SPLINE
SPL {X  -148.173, Y  +313.009, Z    +0.000, E1   +35.624, E3 +294907.954}
SPL {X  -159.343, Y  +347.032, Z    +0.000, E1   +21.245, E3 +294911.798}
SPL {X  -161.787, Y  +362.186, Z    +0.000, E1   +13.182, E3 +294912.994}
SPL {X  -162.692, Y  +374.052, Z    +0.000, E1    +6.208, E3 +294912.840}
SPL {X  -162.820, Y  +381.030, Z    +0.000, E1    +1.454, E3 +294913.019}
SPL {X  -162.820, Y  +384.274, Z    +0.000, E1    -1.205, E3 +294912.738}
SPL {X  -162.820, Y  +388.271, Z    +0.000, E1    -5.458, E3 +294912.730}
SPL {X  -162.820, Y  +394.827, Z    +0.000, E1   -13.677, E3 +294912.420}
SPL {X  -162.820, Y  +402.977, Z    +0.000, E1   -24.772, E3 +294912.702}
SPL {X  -162.820, Y  +413.615, Z    +0.000, E1   -37.560, E3 +294912.493}
SPL {X  -162.820, Y  +452.521, Z    +0.000, E1   -56.942, E3 +294926.785}
SPL {X  -162.820, Y  +459.967, Z    +0.000, E1   -57.801, E3 +294932.081}
SPL {X  -162.820, Y  +525.017, Z    +0.000, E1   -58.379, E3 +295000.199}
ENDSPLINE

SPLINE
SPL {X  -162.820, Y  +515.796, Z    +0.000, E1   -54.952, E3 +295009.306}
ENDSPLINE

SPLINE
SPL {X  -162.820, Y  +522.537, Z    +0.000, E1   -55.218, E3 +295017.481}
SPL {X  -162.820, Y  +529.742, Z    +0.000, E1   -55.146, E3 +295028.408}
SPL {X  -162.820, Y  +538.383, Z    +0.000, E1   -55.306, E3 +295039.860}
SPL {X  -162.820, Y  +544.790, Z    +0.000, E1   -55.066, E3 +295050.660}
SPL {X  -162.820, Y  +552.981, Z    +0.000, E1   -55.286, E3 +295061.122}
SPL {X  -162.820, Y  +560.767, Z    +0.000, E1   -55.137, E3 +295073.431}
SPL {X  -162.820, Y  +570.590, Z    +0.000, E1   -55.270, E3 +295086.765}
SPL {X  -162.820, Y  +580.865, Z    +0.000, E1   -55.132, E3 +295102.722}
SPL {X  -162.820, Y  +591.604, Z    +0.000, E1   -55.202, E3 +295117.659}
SPL {X  -162.820, Y  +600.465, Z    +0.000, E1   -55.218, E3 +295130.447}
SPL {X  -162.820, Y  +609.951, Z    +0.000, E1   -55.211, E3 +295144.195}
SPL {X  -162.820, Y  +618.960, Z    +0.000, E1   -55.186, E3 +295157.415}
SPL {X  -162.820, Y  +627.322, Z    +0.000, E1   -55.201, E3 +295169.350}
SPL {X  -162.820, Y  +634.693, Z    +0.000, E1   -55.198, E3 +295180.067}
SPL {X  -162.820, Y  +642.452, Z    +0.000, E1   -55.141, E3 +295191.674}
SPL {X  -162.820, Y  +649.370, Z    +0.000, E1   -55.160, E3 +295201.530}
SPL {X  -162.820, Y  +658.542, Z    +0.000, E1   -55.251, E3 +295214.409}
SPL {X  -162.820, Y  +668.534, Z    +0.000, E1   -55.182, E3 +295229.204}
SPL {X  -162.763, Y  +677.803, Z    +0.000, E1   -55.175, E3 +295242.710}
SPL {X  -162.314, Y  +686.325, Z    +0.000, E1   -55.173, E3 +295254.990}
SPL {X  -161.784, Y  +691.841, Z    +0.000, E1   -55.010, E3 +295263.952}
SPL {X  -161.070, Y  +697.305, Z    +0.000, E1   -54.828, E3 +295273.030}
SPL {X  -159.751, Y  +704.965, Z    +0.000, E1   -54.697, E3 +295285.016}
SPL {X  -158.271, Y  +711.718, Z    +0.000, E1   -54.504, E3 +295295.825}
SPL {X  -157.115, Y  +716.223, Z    +0.000, E1   -54.227, E3 +295304.017}
SPL {X  -155.622, Y  +721.376, Z    +0.000, E1   -53.849, E3 +295313.617}
SPL {X  -153.323, Y  +728.294, Z    +0.000, E1   -53.618, E3 +295325.090}
SPL {X  -150.606, Y  +735.372, Z    +0.000, E1   -53.091, E3 +295338.086}
SPL {X  -148.712, Y  +739.795, Z    +0.000, E1   -52.656, E3 +295346.649}
SPL {X  -146.885, Y  +743.751, Z    +0.000, E1   -52.544, E3 +295352.922}
SPL {X  -144.373, Y  +748.778, Z    +0.000, E1   -52.887, E3 +295358.385}
SPL {X  -137.947, Y  +759.993, Z    +0.000, E1   -55.381, E3 +295361.495}
SPL {X  -123.111, Y  +780.056, Z    +0.000, E1   -48.144, E3 +295460.630}
ENDSPLINE

SPLINE
SPL {X  -146.599, Y  +744.345, Z    +0.000, E1   -36.661, E3 +295545.633}
SPL {X  -158.886, Y  +709.076, Z    +0.000, E1   -22.176, E3 +295549.505}
SPL {X  -161.886, Y  +690.913, Z    +0.000, E1   -12.672, E3 +295554.140}
SPL {X  -162.573, Y  +682.458, Z    +0.000, E1    -7.683, E3 +295553.641}
SPL {X  -162.817, Y  +674.426, Z    +0.000, E1    -2.573, E3 +295553.359}
SPL {X  -162.820, Y  +670.554, Z    +0.000, E1    +0.472, E3 +295552.983}
SPL {X  -162.820, Y  +667.789, Z    +0.000, E1    +3.144, E3 +295553.005}
SPL {X  -162.820, Y  +664.083, Z    +0.000, E1    +7.387, E3 +295552.897}
SPL {X  -162.820, Y  +659.344, Z    +0.000, E1   +13.535, E3 +295552.460}
SPL {X  -162.820, Y  +653.403, Z    +0.000, E1   +21.415, E3 +295552.875}
SPL {X  -162.820, Y  +642.162, Z    +0.000, E1   +35.510, E3 +295552.187}
SPL {X  -162.820, Y  +598.675, Z    +0.000, E1   +56.845, E3 +295569.500}
SPL {X  -162.820, Y  +543.175, Z    +0.000, E1   +54.504, E3 +295645.354}
SPL {X  -162.820, Y  +538.115, Z    +0.000, E1   +53.658, E3 +295658.406}
SPL {X  -162.820, Y  +527.429, Z    +0.000, E1   +53.760, E3 +295674.135}
SPL {X  -162.820, Y  +518.365, Z    +0.000, E1   +53.683, E3 +295688.393}
SPL {X  -162.820, Y  +510.654, Z    +0.000, E1   +53.658, E3 +295700.392}
SPL {X  -162.820, Y  +501.304, Z    +0.000, E1   +53.758, E3 +295714.081}
SPL {X  -162.820, Y  +493.008, Z    +0.000, E1   +53.586, E3 +295727.856}
SPL {X  -162.820, Y  +484.615, Z    +0.000, E1   +53.726, E3 +295739.787}
ENDSPLINE

SPLINE
SPL {X  -162.820, Y  +492.996, Z    +0.000, E1   +49.430, E3 +295752.333}
ENDSPLINE

SPLINE
SPL {X  -162.820, Y  +486.578, Z    +0.000, E1   +49.194, E3 +295765.136}
SPL {X  -162.820, Y  +476.731, Z    +0.000, E1   +50.039, E3 +295777.558}
SPL {X  -162.820, Y  +466.442, Z    +0.000, E1   +50.873, E3 +295790.227}
SPL {X  -162.820, Y  +458.457, Z    +0.000, E1   +51.401, E3 +295800.366}
SPL {X  -162.820, Y  +452.070, Z    +0.000, E1   +52.035, E3 +295807.002}
SPL {X  -162.820, Y  +442.466, Z    +0.000, E1   +52.743, E3 +295818.214}
SPL {X  -162.820, Y  +429.602, Z    +0.000, E1   +53.907, E3 +295830.916}
SPL {X  -162.820, Y  +419.900, Z    +0.000, E1   +54.598, E3 +295841.168}
SPL {X  -162.820, Y  +411.092, Z    +0.000, E1   +54.552, E3 +295854.688}
SPL {X  -162.820, Y  +400.244, Z    +0.000, E1   +54.630, E3 +295870.155}
SPL {X  -162.820, Y  +392.496, Z    +0.000, E1   +54.734, E3 +295880.856}
SPL {X  -162.820, Y  +387.085, Z    +0.000, E1   +54.699, E3 +295889.083}
SPL {X  -162.820, Y  +380.650, Z    +0.000, E1   +54.601, E3 +295899.179}
SPL {X  -162.727, Y  +374.992, Z    +0.000, E1   +54.549, E3 +295907.861}
SPL {X  -162.373, Y  +368.447, Z    +0.000, E1   +54.597, E3 +295917.293}
SPL {X  -161.939, Y  +363.587, Z    +0.000, E1   +54.355, E3 +295925.905}
SPL {X  -161.062, Y  +356.641, Z    +0.000, E1   +54.440, E3 +295935.778}
SPL {X  -159.761, Y  +349.086, Z    +0.000, E1   +54.132, E3 +295948.799}
SPL {X  -158.033, Y  +341.310, Z    +0.000, E1   +53.819, E3 +295962.189}
SPL {X  -156.195, Y  +334.528, Z    +0.000, E1   +53.534, E3 +295973.755}
SPL {X  -154.120, Y  +327.988, Z    +0.000, E1   +53.171, E3 +295985.612}
SPL {X  -151.310, Y  +320.369, Z    +0.000, E1   +52.706, E3 +295999.327}
SPL {X  -148.923, Y  +314.679, Z    +0.000, E1   +52.172, E3 +296010.411}
SPL {X  -146.846, Y  +310.168, Z    +0.000, E1   +51.697, E3 +296019.473}
SPL {X  -140.627, Y  +298.437, Z    +0.000, E1   +54.251, E3 +296023.731}
SPL {X  -122.064, Y  +272.747, Z    +0.000, E1   +48.156, E3 +296129.257}
ENDSPLINE

SPLINE
SPL {X  -148.173, Y  +313.009, Z    +0.000, E1   +35.624, E3 +296212.302}
SPL {X  -158.289, Y  +342.356, Z    +0.000, E1   +23.452, E3 +296215.292}
SPL {X  -161.301, Y  +358.312, Z    +0.000, E1   +15.384, E3 +296217.249}
SPL {X  -162.692, Y  +374.052, Z    +0.000, E1    +6.208, E3 +296217.188}
SPL {X  -162.820, Y  +381.030, Z    +0.000, E1    +1.454, E3 +296217.366}
SPL {X  -162.820, Y  +384.274, Z    +0.000, E1    -1.205, E3 +296217.086}
SPL {X  -162.820, Y  +388.271, Z    +0.000, E1    -5.458, E3 +296217.078}
SPL {X  -162.820, Y  +394.827, Z    +0.000, E1   -13.677, E3 +296216.768}
SPL {X  -162.820, Y  +402.977, Z    +0.000, E1   -24.772, E3 +296217.050}
SPL {X  -162.820, Y  +413.615, Z    +0.000, E1   -37.560, E3 +296216.841}
SPL {X  -162.820, Y  +456.390, Z    +0.000, E1   -57.415, E3 +296233.882}
SPL {X  -162.820, Y  +525.017, Z    +0.000, E1   -58.379, E3 +296304.547}
ENDSPLINE

SPLINE
SPL {X  -162.820, Y  +520.266, Z    +0.000, E1   -55.155, E3 +296319.039}
ENDSPLINE

SPLINE
SPL {X  -162.820, Y  +529.742, Z    +0.000, E1   -55.146, E3 +296332.755}
SPL {X  -162.820, Y  +538.383, Z    +0.000, E1   -55.306, E3 +296344.208}
SPL {X  -162.820, Y  +544.790, Z    +0.000, E1   -55.066, E3 +296355.008}
SPL {X  -162.820, Y  +555.105, Z    +0.000, E1   -55.222, E3 +296369.128}
SPL {X  -162.820, Y  +563.355, Z    +0.000, E1   -55.172, E3 +296381.195}
SPL {X  -162.820, Y  +570.590, Z    +0.000, E1   -55.270, E3 +296391.113}
SPL {X  -162.820, Y  +580.865, Z    +0.000, E1   -55.132, E3 +296407.070}
SPL {X  -162.820, Y  +591.604, Z    +0.000, E1   -55.202, E3 +296422.007}
SPL {X  -162.820, Y  +600.465, Z    +0.000, E1   -55.218, E3 +296434.795}
SPL {X  -162.820, Y  +609.951, Z    +0.000, E1   -55.211, E3 +296448.543}
SPL {X  -162.820, Y  +618.960, Z    +0.000, E1   -55.186, E3 +296461.763}
SPL {X  -162.820, Y  +627.322, Z    +0.000, E1   -55.201, E3 +296473.698}
SPL {X  -162.820, Y  +634.693, Z    +0.000, E1   -55.198, E3 +296484.415}
SPL {X  -162.820, Y  +642.452, Z    +0.000, E1   -55.141, E3 +296496.021}
SPL {X  -162.820, Y  +649.370, Z    +0.000, E1   -55.160, E3 +296505.878}
SPL {X  -162.820, Y  +658.542, Z    +0.000, E1   -55.251, E3 +296518.757}
SPL {X  -162.820, Y  +668.534, Z    +0.000, E1   -55.182, E3 +296533.552}
SPL {X  -162.763, Y  +677.803, Z    +0.000, E1   -55.175, E3 +296547.058}
SPL {X  -162.084, Y  +688.960, Z    +0.000, E1   -55.150, E3 +296563.513}
SPL {X  -161.070, Y  +697.305, Z    +0.000, E1   -54.828, E3 +296577.378}
SPL {X  -159.751, Y  +704.965, Z    +0.000, E1   -54.697, E3 +296589.364}
SPL {X  -158.271, Y  +711.718, Z    +0.000, E1   -54.504, E3 +296600.173}
SPL {X  -157.115, Y  +716.223, Z    +0.000, E1   -54.227, E3 +296608.364}
SPL {X  -155.622, Y  +721.376, Z    +0.000, E1   -53.849, E3 +296617.964}
SPL {X  -153.323, Y  +728.294, Z    +0.000, E1   -53.618, E3 +296629.437}
SPL {X  -150.606, Y  +735.372, Z    +0.000, E1   -53.091, E3 +296642.434}
SPL {X  -148.712, Y  +739.795, Z    +0.000, E1   -52.656, E3 +296650.997}
SPL {X  -146.885, Y  +743.751, Z    +0.000, E1   -52.544, E3 +296657.270}
SPL {X  -144.373, Y  +748.778, Z    +0.000, E1   -52.887, E3 +296662.733}
SPL {X  -137.947, Y  +759.993, Z    +0.000, E1   -55.381, E3 +296665.842}
SPL {X  -123.111, Y  +780.056, Z    +0.000, E1   -48.144, E3 +296764.978}
ENDSPLINE

SPLINE
SPL {X  -146.599, Y  +744.345, Z    +0.000, E1   -36.661, E3 +296849.981}
SPL {X  -158.886, Y  +709.076, Z    +0.000, E1   -22.176, E3 +296853.853}
SPL {X  -161.886, Y  +690.913, Z    +0.000, E1   -12.672, E3 +296858.488}
SPL {X  -162.700, Y  +679.756, Z    +0.000, E1    -6.060, E3 +296857.697}
SPL {X  -162.820, Y  +673.439, Z    +0.000, E1    -1.797, E3 +296857.799}
SPL {X  -162.820, Y  +670.554, Z    +0.000, E1    +0.472, E3 +296857.331}
SPL {X  -162.820, Y  +667.789, Z    +0.000, E1    +3.144, E3 +296857.353}
SPL {X  -162.820, Y  +664.083, Z    +0.000, E1    +7.387, E3 +296857.244}
SPL {X  -162.820, Y  +659.344, Z    +0.000, E1   +13.535, E3 +296856.808}
SPL {X  -162.820, Y  +653.403, Z    +0.000, E1   +21.415, E3 +296857.223}
SPL {X  -162.820, Y  +642.162, Z    +0.000, E1   +35.510, E3 +296856.535}
SPL {X  -162.820, Y  +598.675, Z    +0.000, E1   +56.845, E3 +296873.848}
SPL {X  -162.820, Y  +542.287, Z    +0.000, E1   +54.257, E3 +296952.751}
SPL {X  -162.820, Y  +533.839, Z    +0.000, E1   +53.682, E3 +296969.172}
SPL {X  -162.820, Y  +525.300, Z    +0.000, E1   +53.701, E3 +296981.947}
SPL {X  -162.820, Y  +518.365, Z    +0.000, E1   +53.683, E3 +296992.741}
SPL {X  -162.820, Y  +508.465, Z    +0.000, E1   +53.706, E3 +297007.956}
SPL {X  -162.820, Y  +499.206, Z    +0.000, E1   +53.779, E3 +297021.395}
SPL {X  -162.820, Y  +493.008, Z    +0.000, E1   +53.586, E3 +297032.204}
SPL {X  -162.820, Y  +485.759, Z    +0.000, E1   +53.138, E3 +297046.211}
ENDSPLINE

SPLINE
SPL {X  -162.820, Y  +494.645, Z    +0.000, E1   +48.544, E3 +297058.687}
ENDSPLINE

SPLINE
SPL {X  -162.820, Y  +486.578, Z    +0.000, E1   +49.194, E3 +297069.483}
SPL {X  -162.820, Y  +476.731, Z    +0.000, E1   +50.039, E3 +297081.906}
SPL {X  -162.820, Y  +466.442, Z    +0.000, E1   +50.873, E3 +297094.575}
SPL {X  -162.820, Y  +458.457, Z    +0.000, E1   +51.401, E3 +297104.714}
SPL {X  -162.820, Y  +452.070, Z    +0.000, E1   +52.035, E3 +297111.349}
SPL {X  -162.820, Y  +442.466, Z    +0.000, E1   +52.743, E3 +297122.562}
SPL {X  -162.820, Y  +429.602, Z    +0.000, E1   +53.907, E3 +297135.264}
SPL {X  -162.820, Y  +419.900, Z    +0.000, E1   +54.598, E3 +297145.516}
SPL {X  -162.820, Y  +411.092, Z    +0.000, E1   +54.552, E3 +297159.036}
SPL {X  -162.820, Y  +400.244, Z    +0.000, E1   +54.630, E3 +297174.503}
SPL {X  -162.820, Y  +389.249, Z    +0.000, E1   +54.752, E3 +297190.082}
SPL {X  -162.799, Y  +377.862, Z    +0.000, E1   +54.622, E3 +297207.712}
SPL {X  -162.373, Y  +368.447, Z    +0.000, E1   +54.597, E3 +297221.641}
SPL {X  -161.939, Y  +363.587, Z    +0.000, E1   +54.355, E3 +297230.253}
SPL {X  -161.062, Y  +356.641, Z    +0.000, E1   +54.440, E3 +297240.126}
SPL {X  -159.761, Y  +349.086, Z    +0.000, E1   +54.132, E3 +297253.147}
SPL {X  -158.451, Y  +343.033, Z    +0.000, E1   +53.828, E3 +297263.824}
SPL {X  -156.619, Y  +335.993, Z    +0.000, E1   +53.639, E3 +297275.470}
SPL {X  -154.959, Y  +330.520, Z    +0.000, E1   +53.198, E3 +297285.895}
SPL {X  -152.785, Y  +324.223, Z    +0.000, E1   +52.975, E3 +297296.568}
SPL {X  -150.663, Y  +318.766, Z    +0.000, E1   +52.574, E3 +297306.601}
SPL {X  -148.923, Y  +314.679, Z    +0.000, E1   +52.172, E3 +297314.759}
SPL {X  -146.846, Y  +310.168, Z    +0.000, E1   +51.697, E3 +297323.820}
SPL {X  -140.627, Y  +298.437, Z    +0.000, E1   +54.251, E3 +297328.079}
SPL {X  -121.787, Y  +272.434, Z    +0.000, E1   +49.053, E3 +297418.440}
ENDSPLINE

SPLINE
SPL {X  -122.346, Y  +273.067, Z    +0.000, E1   +47.776, E3 +297439.631}
SPL {X  -148.173, Y  +313.009, Z    +0.000, E1   +35.624, E3 +297516.650}
SPL {X  -159.343, Y  +347.032, Z    +0.000, E1   +21.245, E3 +297520.494}
SPL {X  -161.787, Y  +362.186, Z    +0.000, E1   +13.182, E3 +297521.689}
SPL {X  -162.692, Y  +374.052, Z    +0.000, E1    +6.208, E3 +297521.535}
SPL {X  -162.820, Y  +382.143, Z    +0.000, E1    +0.693, E3 +297521.670}
SPL {X  -162.820, Y  +385.887, Z    +0.000, E1    -2.819, E3 +297521.342}
SPL {X  -162.820, Y  +389.383, Z    +0.000, E1    -6.871, E3 +297521.409}
SPL {X  -162.820, Y  +393.153, Z    +0.000, E1   -11.600, E3 +297521.303}
SPL {X  -162.820, Y  +400.748, Z    +0.000, E1   -21.791, E3 +297521.094}
SPL {X  -162.820, Y  +413.615, Z    +0.000, E1   -37.560, E3 +297521.189}
SPL {X  -162.820, Y  +456.390, Z    +0.000, E1   -57.415, E3 +297538.230}
SPL {X  -162.820, Y  +525.017, Z    +0.000, E1   -58.379, E3 +297608.895}
ENDSPLINE

SPLINE
SPL {X  -162.820, Y  +520.266, Z    +0.000, E1   -55.155, E3 +297623.387}
ENDSPLINE

SPLINE
SPL {X  -162.820, Y  +529.742, Z    +0.000, E1   -55.146, E3 +297637.103}
SPL {X  -162.820, Y  +538.383, Z    +0.000, E1   -55.306, E3 +297648.555}
SPL {X  -162.820, Y  +544.790, Z    +0.000, E1   -55.066, E3 +297659.356}
SPL {X  -162.820, Y  +552.981, Z    +0.000, E1   -55.286, E3 +297669.818}
SPL {X  -162.820, Y  +560.767, Z    +0.000, E1   -55.137, E3 +297682.126}
SPL {X  -162.820, Y  +570.590, Z    +0.000, E1   -55.270, E3 +297695.461}
SPL {X  -162.820, Y  +577.946, Z    +0.000, E1   -55.110, E3 +297707.098}
SPL {X  -162.820, Y  +583.981, Z    +0.000, E1   -55.057, E3 +297716.181}
SPL {X  -162.820, Y  +591.604, Z    +0.000, E1   -55.202, E3 +297726.355}
SPL {X  -162.820, Y  +600.465, Z    +0.000, E1   -55.218, E3 +297739.143}
SPL {X  -162.820, Y  +609.951, Z    +0.000, E1   -55.211, E3 +297752.891}
SPL {X  -162.820, Y  +618.960, Z    +0.000, E1   -55.186, E3 +297766.111}
SPL {X  -162.820, Y  +627.322, Z    +0.000, E1   -55.201, E3 +297778.046}
SPL {X  -162.820, Y  +634.693, Z    +0.000, E1   -55.198, E3 +297788.763}
SPL {X  -162.820, Y  +642.452, Z    +0.000, E1   -55.141, E3 +297800.369}
SPL {X  -162.820, Y  +652.837, Z    +0.000, E1   -55.281, E3 +297814.637}
SPL {X  -162.820, Y  +660.849, Z    +0.000, E1   -55.101, E3 +297827.186}
SPL {X  -162.820, Y  +668.534, Z    +0.000, E1   -55.182, E3 +297837.900}
SPL {X  -162.763, Y  +677.803, Z    +0.000, E1   -55.175, E3 +297851.406}
SPL {X  -162.084, Y  +688.960, Z    +0.000, E1   -55.150, E3 +297867.861}
SPL {X  -161.070, Y  +697.305, Z    +0.000, E1   -54.828, E3 +297881.726}
SPL {X  -159.751, Y  +704.965, Z    +0.000, E1   -54.697, E3 +297893.712}
SPL {X  -158.271, Y  +711.718, Z    +0.000, E1   -54.504, E3 +297904.521}
SPL {X  -157.115, Y  +716.223, Z    +0.000, E1   -54.227, E3 +297912.712}
SPL {X  -154.825, Y  +723.894, Z    +0.000, E1   -53.830, E3 +297926.252}
SPL {X  -152.160, Y  +731.445, Z    +0.000, E1   -53.336, E3 +297939.795}
SPL {X  -150.059, Y  +736.687, Z    +0.000, E1   -53.023, E3 +297948.961}
SPL {X  -147.746, Y  +741.922, Z    +0.000, E1   -52.631, E3 +297958.668}
SPL {X  -144.373, Y  +748.778, Z    +0.000, E1   -52.887, E3 +297967.081}
SPL {X  -137.947, Y  +759.993, Z    +0.000, E1   -55.381, E3 +297970.190}
SPL {X  -123.111, Y  +780.056, Z    +0.000, E1   -48.144, E3 +298069.326}
ENDSPLINE

SPLINE
SPL {X  -146.599, Y  +744.345, Z    +0.000, E1   -36.661, E3 +298154.329}
SPL {X  -158.886, Y  +709.076, Z    +0.000, E1   -22.176, E3 +298158.201}
SPL {X  -161.886, Y  +690.913, Z    +0.000, E1   -12.672, E3 +298162.835}
SPL {X  -162.700, Y  +679.756, Z    +0.000, E1    -6.060, E3 +298162.045}
SPL {X  -162.820, Y  +673.439, Z    +0.000, E1    -1.797, E3 +298162.146}
SPL {X  -162.820, Y  +670.554, Z    +0.000, E1    +0.472, E3 +298161.679}
SPL {X  -162.820, Y  +667.789, Z    +0.000, E1    +3.144, E3 +298161.701}
SPL {X  -162.820, Y  +664.083, Z    +0.000, E1    +7.387, E3 +298161.592}
SPL {X  -162.820, Y  +659.344, Z    +0.000, E1   +13.535, E3 +298161.156}
SPL {X  -162.820, Y  +653.403, Z    +0.000, E1   +21.415, E3 +298161.571}
SPL {X  -162.820, Y  +642.162, Z    +0.000, E1   +35.510, E3 +298160.883}
SPL {X  -162.820, Y  +598.675, Z    +0.000, E1   +56.845, E3 +298178.195}
SPL {X  -162.820, Y  +543.175, Z    +0.000, E1   +54.504, E3 +298254.050}
SPL {X  -162.820, Y  +538.115, Z    +0.000, E1   +53.658, E3 +298267.101}
SPL {X  -162.820, Y  +527.429, Z    +0.000, E1   +53.760, E3 +298282.831}
SPL {X  -162.820, Y  +518.365, Z    +0.000, E1   +53.683, E3 +298297.089}
SPL {X  -162.820, Y  +510.654, Z    +0.000, E1   +53.658, E3 +298309.088}
SPL {X  -162.820, Y  +501.304, Z    +0.000, E1   +53.758, E3 +298322.776}
SPL {X  -162.820, Y  +493.008, Z    +0.000, E1   +53.586, E3 +298336.552}
SPL {X  -162.820, Y  +484.615, Z    +0.000, E1   +53.726, E3 +298348.482}
ENDSPLINE

SPLINE
SPL {X  -162.820, Y  +492.996, Z    +0.000, E1   +49.430, E3 +298361.028}
ENDSPLINE

SPLINE
SPL {X  -162.820, Y  +486.578, Z    +0.000, E1   +49.194, E3 +298373.831}
SPL {X  -162.820, Y  +476.731, Z    +0.000, E1   +50.039, E3 +298386.254}
SPL {X  -162.820, Y  +466.442, Z    +0.000, E1   +50.873, E3 +298398.922}
SPL {X  -162.820, Y  +455.624, Z    +0.000, E1   +51.698, E3 +298411.994}
SPL {X  -162.820, Y  +444.568, Z    +0.000, E1   +52.608, E3 +298424.306}
SPL {X  -162.820, Y  +432.435, Z    +0.000, E1   +53.605, E3 +298437.189}
SPL {X  -162.820, Y  +419.875, Z    +0.000, E1   +54.604, E3 +298449.864}
SPL {X  -162.820, Y  +414.181, Z    +0.000, E1   +54.446, E3 +298459.298}
SPL {X  -162.820, Y  +407.616, Z    +0.000, E1   +54.585, E3 +298468.132}
SPL {X  -162.820, Y  +400.244, Z    +0.000, E1   +54.630, E3 +298478.851}
SPL {X  -162.820, Y  +389.249, Z    +0.000, E1   +54.752, E3 +298494.430}
SPL {X  -162.820, Y  +380.650, Z    +0.000, E1   +54.601, E3 +298507.875}
SPL {X  -162.727, Y  +374.992, Z    +0.000, E1   +54.549, E3 +298516.557}
SPL {X  -162.373, Y  +368.447, Z    +0.000, E1   +54.597, E3 +298525.989}
SPL {X  -161.939, Y  +363.587, Z    +0.000, E1   +54.355, E3 +298534.601}
SPL {X  -161.062, Y  +356.641, Z    +0.000, E1   +54.440, E3 +298544.474}
SPL {X  -159.761, Y  +349.086, Z    +0.000, E1   +54.132, E3 +298557.495}
SPL {X  -158.033, Y  +341.310, Z    +0.000, E1   +53.819, E3 +298570.885}
SPL {X  -155.608, Y  +332.578, Z    +0.000, E1   +53.425, E3 +298586.156}
SPL {X  -152.785, Y  +324.223, Z    +0.000, E1   +52.975, E3 +298600.916}
SPL {X  -150.663, Y  +318.766, Z    +0.000, E1   +52.574, E3 +298610.949}
SPL {X  -148.923, Y  +314.679, Z    +0.000, E1   +52.172, E3 +298619.107}
SPL {X  -146.846, Y  +310.168, Z    +0.000, E1   +51.697, E3 +298628.168}
SPL {X  -140.627, Y  +298.437, Z    +0.000, E1   +54.251, E3 +298632.427}
SPL {X  -122.064, Y  +272.747, Z    +0.000, E1   +48.156, E3 +298737.952}
ENDSPLINE

SPLINE
SPL {X  -148.173, Y  +313.009, Z    +0.000, E1   +35.624, E3 +298820.998}
SPL {X  -159.343, Y  +347.032, Z    +0.000, E1   +21.245, E3 +298824.842}
SPL {X  -162.355, Y  +368.197, Z    +0.000, E1    +9.799, E3 +298826.010}
SPL {X  -162.819, Y  +380.071, Z    +0.000, E1    +2.240, E3 +298826.005}
SPL {X  -162.820, Y  +384.274, Z    +0.000, E1    -1.205, E3 +298825.781}
SPL {X  -162.820, Y  +388.271, Z    +0.000, E1    -5.458, E3 +298825.774}
SPL {X  -162.820, Y  +394.827, Z    +0.000, E1   -13.677, E3 +298825.464}
SPL {X  -162.820, Y  +402.977, Z    +0.000, E1   -24.772, E3 +298825.746}
SPL {X  -162.820, Y  +413.615, Z    +0.000, E1   -37.560, E3 +298825.536}
SPL {X  -162.820, Y  +456.390, Z    +0.000, E1   -57.415, E3 +298842.578}
SPL {X  -162.820, Y  +525.017, Z    +0.000, E1   -58.379, E3 +298913.242}
ENDSPLINE

SPLINE
SPL {X  -162.820, Y  +515.796, Z    +0.000, E1   -54.952, E3 +298922.349}
ENDSPLINE

SPLINE
SPL {X  -162.820, Y  +522.537, Z    +0.000, E1   -55.218, E3 +298930.524}
SPL {X  -162.820, Y  +529.742, Z    +0.000, E1   -55.146, E3 +298941.451}
SPL {X  -162.820, Y  +538.383, Z    +0.000, E1   -55.306, E3 +298952.903}
SPL {X  -162.820, Y  +544.790, Z    +0.000, E1   -55.066, E3 +298963.703}
SPL {X  -162.820, Y  +555.105, Z    +0.000, E1   -55.222, E3 +298977.824}
SPL {X  -162.820, Y  +563.355, Z    +0.000, E1   -55.172, E3 +298989.891}
SPL {X  -162.820, Y  +570.590, Z    +0.000, E1   -55.270, E3 +298999.808}
SPL {X  -162.820, Y  +580.865, Z    +0.000, E1   -55.132, E3 +299015.765}
SPL {X  -162.820, Y  +594.246, Z    +0.000, E1   -55.310, E3 +299033.964}
SPL {X  -162.820, Y  +601.811, Z    +0.000, E1   -55.027, E3 +299046.492}
SPL {X  -162.820, Y  +609.951, Z    +0.000, E1   -55.211, E3 +299057.238}
SPL {X  -162.820, Y  +618.960, Z    +0.000, E1   -55.186, E3 +299070.459}
SPL {X  -162.820, Y  +627.322, Z    +0.000, E1   -55.201, E3 +299082.394}
SPL {X  -162.820, Y  +634.693, Z    +0.000, E1   -55.198, E3 +299093.110}
SPL {X  -162.820, Y  +642.452, Z    +0.000, E1   -55.141, E3 +299104.717}
SPL {X  -162.820, Y  +649.370, Z    +0.000, E1   -55.160, E3 +299114.574}
SPL {X  -162.820, Y  +658.542, Z    +0.000, E1   -55.251, E3 +299127.452}
SPL {X  -162.820, Y  +671.259, Z    +0.000, E1   -55.266, E3 +299145.830}
SPL {X  -162.498, Y  +683.731, Z    +0.000, E1   -55.157, E3 +299164.539}
SPL {X  -161.784, Y  +691.841, Z    +0.000, E1   -55.010, E3 +299176.996}
SPL {X  -161.070, Y  +697.305, Z    +0.000, E1   -54.828, E3 +299186.074}
SPL {X  -159.751, Y  +704.965, Z    +0.000, E1   -54.697, E3 +299198.060}
SPL {X  -158.271, Y  +711.718, Z    +0.000, E1   -54.504, E3 +299208.868}
SPL {X  -157.115, Y  +716.223, Z    +0.000, E1   -54.227, E3 +299217.060}
SPL {X  -154.825, Y  +723.894, Z    +0.000, E1   -53.830, E3 +299230.600}
SPL {X  -152.160, Y  +731.445, Z    +0.000, E1   -53.336, E3 +299244.142}
SPL {X  -150.059, Y  +736.687, Z    +0.000, E1   -53.023, E3 +299253.308}
SPL {X  -147.746, Y  +741.922, Z    +0.000, E1   -52.631, E3 +299263.016}
SPL {X  -144.373, Y  +748.778, Z    +0.000, E1   -52.887, E3 +299271.428}
SPL {X  -137.947, Y  +759.993, Z    +0.000, E1   -55.381, E3 +299274.538}
SPL {X  -123.111, Y  +780.056, Z    +0.000, E1   -48.144, E3 +299373.674}
ENDSPLINE

SPLINE
SPL {X  -146.599, Y  +744.345, Z    +0.000, E1   -36.661, E3 +299458.677}
SPL {X  -157.185, Y  +715.965, Z    +0.000, E1   -25.340, E3 +299461.727}
SPL {X  -159.997, Y  +703.690, Z    +0.000, E1   -19.457, E3 +299463.055}
SPL {X  -161.886, Y  +690.913, Z    +0.000, E1   -12.672, E3 +299467.183}
SPL {X  -162.700, Y  +679.756, Z    +0.000, E1    -6.060, E3 +299466.392}
SPL {X  -162.820, Y  +673.439, Z    +0.000, E1    -1.797, E3 +299466.494}
SPL {X  -162.820, Y  +670.554, Z    +0.000, E1    +0.472, E3 +299466.027}
SPL {X  -162.820, Y  +667.789, Z    +0.000, E1    +3.144, E3 +299466.048}
SPL {X  -162.820, Y  +664.083, Z    +0.000, E1    +7.387, E3 +299465.940}
SPL {X  -162.820, Y  +659.344, Z    +0.000, E1   +13.535, E3 +299465.504}
SPL {X  -162.820, Y  +653.403, Z    +0.000, E1   +21.415, E3 +299465.918}
SPL {X  -162.820, Y  +642.162, Z    +0.000, E1   +35.510, E3 +299465.231}
SPL {X  -162.820, Y  +598.675, Z    +0.000, E1   +56.845, E3 +299482.543}
SPL {X  -162.820, Y  +543.175, Z    +0.000, E1   +54.504, E3 +299558.398}
SPL {X  -162.820, Y  +538.115, Z    +0.000, E1   +53.658, E3 +299571.449}
SPL {X  -162.820, Y  +527.429, Z    +0.000, E1   +53.760, E3 +299587.179}
SPL {X  -162.820, Y  +518.365, Z    +0.000, E1   +53.683, E3 +299601.437}
SPL {X  -162.820, Y  +510.654, Z    +0.000, E1   +53.658, E3 +299613.436}
SPL {X  -162.820, Y  +501.304, Z    +0.000, E1   +53.758, E3 +299627.124}
SPL {X  -162.820, Y  +493.008, Z    +0.000, E1   +53.586, E3 +299640.899}
SPL {X  -162.820, Y  +484.615, Z    +0.000, E1   +53.726, E3 +299652.830}
ENDSPLINE

SPLINE
SPL {X  -162.820, Y  +492.996, Z    +0.000, E1   +49.430, E3 +299665.376}
ENDSPLINE

SPLINE
SPL {X  -162.820, Y  +486.578, Z    +0.000, E1   +49.194, E3 +299678.179}
SPL {X  -162.820, Y  +476.731, Z    +0.000, E1   +50.039, E3 +299690.602}
SPL {X  -162.820, Y  +466.442, Z    +0.000, E1   +50.873, E3 +299703.270}
SPL {X  -162.820, Y  +455.624, Z    +0.000, E1   +51.698, E3 +299716.341}
SPL {X  -162.820, Y  +444.568, Z    +0.000, E1   +52.608, E3 +299728.654}
SPL {X  -162.820, Y  +432.435, Z    +0.000, E1   +53.605, E3 +299741.537}
SPL {X  -162.820, Y  +419.875, Z    +0.000, E1   +54.604, E3 +299754.211}
SPL {X  -162.820, Y  +414.181, Z    +0.000, E1   +54.446, E3 +299763.646}
SPL {X  -162.820, Y  +407.616, Z    +0.000, E1   +54.585, E3 +299772.480}
SPL {X  -162.820, Y  +400.244, Z    +0.000, E1   +54.630, E3 +299783.198}
SPL {X  -162.820, Y  +389.249, Z    +0.000, E1   +54.752, E3 +299798.777}
SPL {X  -162.799, Y  +377.862, Z    +0.000, E1   +54.622, E3 +299816.408}
SPL {X  -162.373, Y  +368.447, Z    +0.000, E1   +54.597, E3 +299830.337}
SPL {X  -161.939, Y  +363.587, Z    +0.000, E1   +54.355, E3 +299838.949}
SPL {X  -161.062, Y  +356.641, Z    +0.000, E1   +54.440, E3 +299848.822}
SPL {X  -159.761, Y  +349.086, Z    +0.000, E1   +54.132, E3 +299861.843}
SPL {X  -158.451, Y  +343.033, Z    +0.000, E1   +53.828, E3 +299872.520}
SPL {X  -156.619, Y  +335.993, Z    +0.000, E1   +53.639, E3 +299884.166}
SPL {X  -154.120, Y  +327.988, Z    +0.000, E1   +53.171, E3 +299898.656}
SPL {X  -151.310, Y  +320.369, Z    +0.000, E1   +52.706, E3 +299912.370}
SPL {X  -148.923, Y  +314.679, Z    +0.000, E1   +52.172, E3 +299923.455}
SPL {X  -146.846, Y  +310.168, Z    +0.000, E1   +51.697, E3 +299932.516}
SPL {X  -140.627, Y  +298.437, Z    +0.000, E1   +54.251, E3 +299936.775}
SPL {X  -122.064, Y  +272.747, Z    +0.000, E1   +48.156, E3 +300042.300}
ENDSPLINE

SPLINE
SPL {X  -148.173, Y  +313.009, Z    +0.000, E1   +35.624, E3 +300125.346}
SPL {X  -159.343, Y  +347.032, Z    +0.000, E1   +21.245, E3 +300129.189}
SPL {X  -162.355, Y  +368.197, Z    +0.000, E1    +9.799, E3 +300130.358}
SPL {X  -162.819, Y  +380.071, Z    +0.000, E1    +2.240, E3 +300130.353}
SPL {X  -162.820, Y  +383.414, Z    +0.000, E1    -0.499, E3 +300130.316}
SPL {X  -162.820, Y  +385.887, Z    +0.000, E1    -2.819, E3 +300130.038}
SPL {X  -162.820, Y  +389.383, Z    +0.000, E1    -6.871, E3 +300130.105}
SPL {X  -162.820, Y  +393.153, Z    +0.000, E1   -11.600, E3 +300129.999}
SPL {X  -162.820, Y  +400.748, Z    +0.000, E1   -21.791, E3 +300129.790}
SPL {X  -162.820, Y  +413.615, Z    +0.000, E1   -37.560, E3 +300129.884}
SPL {X  -162.820, Y  +456.390, Z    +0.000, E1   -57.415, E3 +300146.926}
SPL {X  -162.820, Y  +525.017, Z    +0.000, E1   -58.379, E3 +300217.590}
ENDSPLINE

SPLINE
SPL {X  -162.820, Y  +515.796, Z    +0.000, E1   -54.952, E3 +300226.697}
ENDSPLINE

SPLINE
SPL {X  -162.820, Y  +522.537, Z    +0.000, E1   -55.218, E3 +300234.872}
SPL {X  -162.820, Y  +529.742, Z    +0.000, E1   -55.146, E3 +300245.799}
SPL {X  -162.820, Y  +538.383, Z    +0.000, E1   -55.306, E3 +300257.251}
SPL {X  -162.820, Y  +544.790, Z    +0.000, E1   -55.066, E3 +300268.051}
SPL {X  -162.820, Y  +555.105, Z    +0.000, E1   -55.222, E3 +300282.172}
SPL {X  -162.820, Y  +563.355, Z    +0.000, E1   -55.172, E3 +300294.238}
SPL {X  -162.820, Y  +570.590, Z    +0.000, E1   -55.270, E3 +300304.156}
SPL {X  -162.820, Y  +580.865, Z    +0.000, E1   -55.132, E3 +300320.113}
SPL {X  -162.820, Y  +591.604, Z    +0.000, E1   -55.202, E3 +300335.050}
SPL {X  -162.820, Y  +600.465, Z    +0.000, E1   -55.218, E3 +300347.839}
SPL {X  -162.820, Y  +609.951, Z    +0.000, E1   -55.211, E3 +300361.586}
SPL {X  -162.820, Y  +618.960, Z    +0.000, E1   -55.186, E3 +300374.806}
SPL {X  -162.820, Y  +627.322, Z    +0.000, E1   -55.201, E3 +300386.742}
SPL {X  -162.820, Y  +634.693, Z    +0.000, E1   -55.198, E3 +300397.458}
SPL {X  -162.820, Y  +642.452, Z    +0.000, E1   -55.141, E3 +300409.065}
SPL {X  -162.820, Y  +649.370, Z    +0.000, E1   -55.160, E3 +300418.922}
SPL {X  -162.820, Y  +658.542, Z    +0.000, E1   -55.251, E3 +300431.800}
SPL {X  -162.820, Y  +671.259, Z    +0.000, E1   -55.266, E3 +300450.177}
SPL {X  -162.498, Y  +683.731, Z    +0.000, E1   -55.157, E3 +300468.887}
SPL {X  -161.784, Y  +691.841, Z    +0.000, E1   -55.010, E3 +300481.344}
SPL {X  -161.070, Y  +697.305, Z    +0.000, E1   -54.828, E3 +300490.422}
SPL {X  -159.751, Y  +704.965, Z    +0.000, E1   -54.697, E3 +300502.408}
SPL {X  -158.271, Y  +711.718, Z    +0.000, E1   -54.504, E3 +300513.216}
SPL {X  -157.115, Y  +716.223, Z    +0.000, E1   -54.227, E3 +300521.408}
SPL {X  -155.622, Y  +721.376, Z    +0.000, E1   -53.849, E3 +300531.008}
SPL {X  -153.323, Y  +728.294, Z    +0.000, E1   -53.618, E3 +300542.481}
SPL {X  -150.606, Y  +735.372, Z    +0.000, E1   -53.091, E3 +300555.478}
SPL {X  -148.712, Y  +739.795, Z    +0.000, E1   -52.656, E3 +300564.040}
SPL {X  -146.885, Y  +743.751, Z    +0.000, E1   -52.544, E3 +300570.314}
SPL {X  -144.373, Y  +748.778, Z    +0.000, E1   -52.887, E3 +300575.776}
SPL {X  -137.947, Y  +759.993, Z    +0.000, E1   -55.381, E3 +300578.886}
SPL {X  -123.111, Y  +780.056, Z    +0.000, E1   -48.144, E3 +300678.022}
ENDSPLINE

SPLINE
SPL {X  -146.599, Y  +744.345, Z    +0.000, E1   -36.661, E3 +300763.025}
SPL {X  -158.886, Y  +709.076, Z    +0.000, E1   -22.176, E3 +300766.897}
SPL {X  -161.886, Y  +690.913, Z    +0.000, E1   -12.672, E3 +300771.531}
SPL {X  -162.573, Y  +682.458, Z    +0.000, E1    -7.683, E3 +300771.032}
SPL {X  -162.817, Y  +674.426, Z    +0.000, E1    -2.573, E3 +300770.750}
SPL {X  -162.820, Y  +670.554, Z    +0.000, E1    +0.472, E3 +300770.375}
SPL {X  -162.820, Y  +667.789, Z    +0.000, E1    +3.144, E3 +300770.396}
SPL {X  -162.820, Y  +664.083, Z    +0.000, E1    +7.387, E3 +300770.288}
SPL {X  -162.820, Y  +659.344, Z    +0.000, E1   +13.535, E3 +300769.852}
SPL {X  -162.820, Y  +653.403, Z    +0.000, E1   +21.415, E3 +300770.266}
SPL {X  -162.820, Y  +642.162, Z    +0.000, E1   +35.510, E3 +300769.579}
SPL {X  -162.820, Y  +598.675, Z    +0.000, E1   +56.845, E3 +300786.891}
SPL {X  -162.820, Y  +543.175, Z    +0.000, E1   +54.504, E3 +300862.746}
SPL {X  -162.820, Y  +538.115, Z    +0.000, E1   +53.658, E3 +300875.797}
SPL {X  -162.820, Y  +527.429, Z    +0.000, E1   +53.760, E3 +300891.527}
SPL {X  -162.820, Y  +518.365, Z    +0.000, E1   +53.683, E3 +300905.784}
SPL {X  -162.820, Y  +510.654, Z    +0.000, E1   +53.658, E3 +300917.783}
SPL {X  -162.820, Y  +501.304, Z    +0.000, E1   +53.758, E3 +300931.472}
SPL {X  -162.820, Y  +493.008, Z    +0.000, E1   +53.586, E3 +300945.247}
SPL {X  -162.820, Y  +484.615, Z    +0.000, E1   +53.726, E3 +300957.178}
ENDSPLINE

SPLINE
SPL {X  -162.820, Y  +492.996, Z    +0.000, E1   +49.430, E3 +300969.724}
ENDSPLINE

SPLINE
SPL {X  -162.820, Y  +486.578, Z    +0.000, E1   +49.194, E3 +300982.527}
SPL {X  -162.820, Y  +476.731, Z    +0.000, E1   +50.039, E3 +300994.950}
SPL {X  -162.820, Y  +466.442, Z    +0.000, E1   +50.873, E3 +301007.618}
SPL {X  -162.820, Y  +455.624, Z    +0.000, E1   +51.698, E3 +301020.689}
SPL {X  -162.820, Y  +444.568, Z    +0.000, E1   +52.608, E3 +301033.002}
SPL {X  -162.820, Y  +432.435, Z    +0.000, E1   +53.605, E3 +301045.885}
SPL {X  -162.820, Y  +419.900, Z    +0.000, E1   +54.598, E3 +301058.560}
ENDSPLINE

SPLINE
SPL {X  -162.820, Y  +430.533, Z    +0.000, E1   +49.727, E3 +301071.537}
ENDSPLINE

SPLINE
SPL {X  -162.820, Y  +420.882, Z    +0.000, E1   +49.790, E3 +301088.174}
SPL {X  -162.820, Y  +411.982, Z    +0.000, E1   +49.786, E3 +301103.857}
SPL {X  -162.820, Y  +402.501, Z    +0.000, E1   +49.838, E3 +301120.282}
SPL {X  -162.820, Y  +393.582, Z    +0.000, E1   +49.779, E3 +301136.280}
SPL {X  -162.820, Y  +386.334, Z    +0.000, E1   +49.739, E3 +301149.217}
SPL {X  -162.801, Y  +377.981, Z    +0.000, E1   +49.798, E3 +301163.739}
SPL {X  -162.415, Y  +369.029, Z    +0.000, E1   +49.751, E3 +301179.725}
SPL {X  -161.760, Y  +361.947, Z    +0.000, E1   +49.515, E3 +301193.564}
SPL {X  -160.828, Y  +355.106, Z    +0.000, E1   +49.536, E3 +301205.480}
SPL {X  -159.832, Y  +349.452, Z    +0.000, E1   +49.188, E3 +301217.452}
SPL {X  -158.863, Y  +344.823, Z    +0.000, E1   +49.020, E3 +301226.501}
SPL {X  -157.695, Y  +339.971, Z    +0.000, E1   +48.934, E3 +301235.597}
SPL {X  -156.136, Y  +334.326, Z    +0.000, E1   +48.578, E3 +301247.563}
SPL {X  -153.956, Y  +327.511, Z    +0.000, E1   +48.205, E3 +301261.685}
SPL {X  -151.316, Y  +320.384, Z    +0.000, E1   +47.734, E3 +301276.689}
SPL {X  -145.123, Y  +306.679, Z    +0.000, E1   +50.518, E3 +301285.504}
SPL {X  -135.207, Y  +289.783, Z    +0.000, E1   +44.101, E3 +301379.018}
ENDSPLINE

SPLINE
SPL {X  -154.528, Y  +329.203, Z    +0.000, E1   +28.834, E3 +301449.380}
SPL {X  -160.380, Y  +352.419, Z    +0.000, E1   +18.163, E3 +301453.740}
SPL {X  -162.149, Y  +365.734, Z    +0.000, E1   +11.090, E3 +301452.348}
SPL {X  -162.754, Y  +375.862, Z    +0.000, E1    +5.134, E3 +301453.185}
SPL {X  -162.820, Y  +382.085, Z    +0.000, E1    +0.928, E3 +301452.874}
SPL {X  -162.820, Y  +386.028, Z    +0.000, E1    -2.328, E3 +301452.598}
SPL {X  -162.820, Y  +389.792, Z    +0.000, E1    -6.211, E3 +301452.530}
SPL {X  -162.820, Y  +394.068, Z    +0.000, E1   -11.043, E3 +301452.647}
SPL {X  -162.820, Y  +398.921, Z    +0.000, E1   -16.945, E3 +301452.701}
SPL {X  -162.820, Y  +409.049, Z    +0.000, E1   -29.128, E3 +301451.510}
SPL {X  -162.820, Y  +444.592, Z    +0.000, E1   -49.032, E3 +301470.519}
SPL {X  -162.820, Y  +458.217, Z    +0.000, E1   -51.268, E3 +301482.465}
SPL {X  -162.820, Y  +501.848, Z    +0.000, E1   -54.235, E3 +301528.832}
ENDSPLINE

SPLINE
SPL {X  -162.820, Y  +498.156, Z    +0.000, E1   -50.986, E3 +301542.382}
ENDSPLINE

SPLINE
SPL {X  -162.820, Y  +499.429, Z    +0.000, E1   -49.453, E3 +301553.740}
SPL {X  -162.820, Y  +507.703, Z    +0.000, E1   -49.462, E3 +301568.655}
SPL {X  -162.820, Y  +516.435, Z    +0.000, E1   -49.526, E3 +301583.624}
SPL {X  -162.820, Y  +523.383, Z    +0.000, E1   -49.407, E3 +301596.811}
SPL {X  -162.820, Y  +532.283, Z    +0.000, E1   -49.462, E3 +301612.413}
SPL {X  -162.820, Y  +541.471, Z    +0.000, E1   -49.456, E3 +301628.791}
SPL {X  -162.820, Y  +548.933, Z    +0.000, E1   -49.456, E3 +301641.980}
SPL {X  -162.820, Y  +553.997, Z    +0.000, E1   -49.325, E3 +301651.783}
SPL {X  -162.820, Y  +560.268, Z    +0.000, E1   -49.531, E3 +301661.741}
SPL {X  -162.820, Y  +564.590, Z    +0.000, E1   -49.361, E3 +301670.441}
SPL {X  -162.820, Y  +570.444, Z    +0.000, E1   -49.421, E3 +301680.593}
SPL {X  -162.820, Y  +577.429, Z    +0.000, E1   -49.474, E3 +301692.707}
SPL {X  -162.820, Y  +585.965, Z    +0.000, E1   -49.447, E3 +301708.281}
SPL {X  -162.820, Y  +594.192, Z    +0.000, E1   -49.325, E3 +301723.524}
SPL {X  -162.820, Y  +600.267, Z    +0.000, E1   -49.443, E3 +301733.612}
SPL {X  -162.820, Y  +606.218, Z    +0.000, E1   -49.464, E3 +301744.159}
SPL {X  -162.820, Y  +612.538, Z    +0.000, E1   -49.488, E3 +301755.210}
SPL {X  -162.820, Y  +617.738, Z    +0.000, E1   -49.301, E3 +301765.647}
SPL {X  -162.820, Y  +624.265, Z    +0.000, E1   -49.443, E3 +301776.442}
SPL {X  -162.820, Y  +632.551, Z    +0.000, E1   -49.478, E3 +301791.211}
SPL {X  -162.820, Y  +641.207, Z    +0.000, E1   -49.420, E3 +301806.854}
SPL {X  -162.820, Y  +649.864, Z    +0.000, E1   -49.433, E3 +301822.332}
SPL {X  -162.820, Y  +658.147, Z    +0.000, E1   -49.491, E3 +301836.599}
SPL {X  -162.820, Y  +663.916, Z    +0.000, E1   -49.371, E3 +301847.589}
SPL {X  -162.820, Y  +669.755, Z    +0.000, E1   -49.387, E3 +301857.913}
SPL {X  -162.807, Y  +675.597, Z    +0.000, E1   -49.472, E3 +301867.816}
SPL {X  -162.632, Y  +681.322, Z    +0.000, E1   -49.345, E3 +301878.827}
SPL {X  -162.228, Y  +687.372, Z    +0.000, E1   -49.294, E3 +301889.914}
SPL {X  -161.723, Y  +692.372, Z    +0.000, E1   -49.172, E3 +301899.544}
SPL {X  -161.009, Y  +697.714, Z    +0.000, E1   -49.214, E3 +301908.828}
SPL {X  -160.313, Y  +701.965, Z    +0.000, E1   -48.932, E3 +301918.041}
SPL {X  -158.980, Y  +708.651, Z    +0.000, E1   -48.774, E3 +301931.081}
SPL {X  -157.477, Y  +714.869, Z    +0.000, E1   -48.424, E3 +301943.955}
SPL {X  -156.071, Y  +719.891, Z    +0.000, E1   -48.264, E3 +301953.832}
SPL {X  -154.661, Y  +724.395, Z    +0.000, E1   -47.951, E3 +301963.513}
SPL {X  -153.094, Y  +728.931, Z    +0.000, E1   -47.705, E3 +301972.950}
SPL {X  -151.300, Y  +733.655, Z    +0.000, E1   -47.339, E3 +301983.259}
SPL {X  -145.669, Y  +746.239, Z    +0.000, E1   -50.198, E3 +301990.035}
SPL {X  -135.084, Y  +764.399, Z    +0.000, E1   -44.787, E3 +302072.939}
ENDSPLINE

SPLINE
SPL {X  -153.038, Y  +729.086, Z    +0.000, E1   -30.522, E3 +302143.646}
SPL {X  -160.383, Y  +701.564, Z    +0.000, E1   -18.145, E3 +302153.682}
SPL {X  -162.078, Y  +689.023, Z    +0.000, E1   -11.510, E3 +302153.220}
SPL {X  -162.685, Y  +680.136, Z    +0.000, E1    -6.379, E3 +302153.509}
SPL {X  -162.820, Y  +672.919, Z    +0.000, E1    -1.752, E3 +302153.548}
SPL {X  -162.820, Y  +669.270, Z    +0.000, E1    +1.140, E3 +302153.030}
SPL {X  -162.820, Y  +666.754, Z    +0.000, E1    +3.396, E3 +302153.599}
SPL {X  -162.820, Y  +662.755, Z    +0.000, E1    +7.521, E3 +302153.389}
SPL {X  -162.820, Y  +657.537, Z    +0.000, E1   +13.540, E3 +302153.059}
SPL {X  -162.820, Y  +650.460, Z    +0.000, E1   +22.200, E3 +302152.490}
SPL {X  -162.820, Y  +637.843, Z    +0.000, E1   +35.051, E3 +302154.566}
SPL {X  -162.820, Y  +595.072, Z    +0.000, E1   +53.652, E3 +302175.287}
SPL {X  -162.820, Y  +560.706, Z    +0.000, E1   +50.482, E3 +302236.196}
ENDSPLINE

SPLINE
SPL {X  -162.820, Y  +560.978, Z    +0.000, E1   +48.448, E3 +302248.281}
ENDSPLINE

SPLINE
SPL {X  -162.820, Y  +552.125, Z    +0.000, E1   +48.477, E3 +302264.386}
SPL {X  -162.820, Y  +545.800, Z    +0.000, E1   +48.334, E3 +302276.828}
SPL {X  -162.820, Y  +538.900, Z    +0.000, E1   +48.334, E3 +302289.743}
SPL {X  -162.820, Y  +530.572, Z    +0.000, E1   +48.392, E3 +302304.793}
SPL {X  -162.820, Y  +524.414, Z    +0.000, E1   +48.297, E3 +302316.676}
SPL {X  -162.820, Y  +516.130, Z    +0.000, E1   +48.458, E3 +302331.260}
SPL {X  -162.820, Y  +508.282, Z    +0.000, E1   +48.307, E3 +302346.516}
SPL {X  -162.820, Y  +502.890, Z    +0.000, E1   +48.309, E3 +302356.442}
ENDSPLINE

SPLINE
SPL {X  -162.820, Y  +517.326, Z    +0.000, E1   +41.232, E3 +302368.707}
ENDSPLINE

SPLINE
SPL {X  -162.820, Y  +507.007, Z    +0.000, E1   +42.470, E3 +302385.385}
SPL {X  -162.820, Y  +496.780, Z    +0.000, E1   +43.573, E3 +302401.640}
SPL {X  -162.820, Y  +488.962, Z    +0.000, E1   +44.342, E3 +302413.907}
SPL {X  -162.820, Y  +481.373, Z    +0.000, E1   +45.107, E3 +302425.392}
SPL {X  -162.820, Y  +473.909, Z    +0.000, E1   +45.743, E3 +302436.904}
SPL {X  -162.820, Y  +465.836, Z    +0.000, E1   +46.727, E3 +302447.195}
SPL {X  -162.820, Y  +457.217, Z    +0.000, E1   +47.671, E3 +302458.233}
SPL {X  -162.820, Y  +449.104, Z    +0.000, E1   +48.459, E3 +302468.702}
SPL {X  -162.820, Y  +440.303, Z    +0.000, E1   +49.204, E3 +302480.339}
SPL {X  -162.820, Y  +430.072, Z    +0.000, E1   +49.865, E3 +302494.641}
SPL {X  -162.820, Y  +423.062, Z    +0.000, E1   +49.728, E3 +302507.634}
SPL {X  -162.820, Y  +416.560, Z    +0.000, E1   +49.816, E3 +302518.615}
SPL {X  -162.820, Y  +410.559, Z    +0.000, E1   +49.727, E3 +302529.671}
SPL {X  -162.820, Y  +405.170, Z    +0.000, E1   +49.772, E3 +302538.872}
SPL {X  -162.820, Y  +398.766, Z    +0.000, E1   +49.793, E3 +302550.160}
SPL {X  -162.820, Y  +391.831, Z    +0.000, E1   +49.801, E3 +302562.206}
SPL {X  -162.820, Y  +386.334, Z    +0.000, E1   +49.739, E3 +302572.294}
SPL {X  -162.820, Y  +381.297, Z    +0.000, E1   +49.665, E3 +302581.565}
SPL {X  -162.709, Y  +374.487, Z    +0.000, E1   +49.773, E3 +302593.090}
SPL {X  -162.299, Y  +367.483, Z    +0.000, E1   +49.784, E3 +302605.232}
SPL {X  -161.760, Y  +361.947, Z    +0.000, E1   +49.515, E3 +302616.641}
SPL {X  -160.828, Y  +355.106, Z    +0.000, E1   +49.536, E3 +302628.557}
SPL {X  -159.832, Y  +349.452, Z    +0.000, E1   +49.188, E3 +302640.529}
SPL {X  -158.863, Y  +344.823, Z    +0.000, E1   +49.020, E3 +302649.578}
SPL {X  -157.695, Y  +339.971, Z    +0.000, E1   +48.934, E3 +302658.674}
SPL {X  -156.496, Y  +335.563, Z    +0.000, E1   +48.599, E3 +302668.251}
SPL {X  -154.894, Y  +330.318, Z    +0.000, E1   +48.380, E3 +302678.794}
SPL {X  -153.352, Y  +325.786, Z    +0.000, E1   +48.028, E3 +302688.551}
SPL {X  -151.316, Y  +320.384, Z    +0.000, E1   +47.734, E3 +302699.766}
SPL {X  -145.123, Y  +306.679, Z    +0.000, E1   +50.518, E3 +302708.581}
SPL {X  -135.207, Y  +289.783, Z    +0.000, E1   +44.101, E3 +302802.095}
ENDSPLINE

SPLINE
SPL {X  -154.528, Y  +329.203, Z    +0.000, E1   +28.834, E3 +302872.456}
SPL {X  -160.380, Y  +352.419, Z    +0.000, E1   +18.163, E3 +302876.817}
SPL {X  -162.408, Y  +368.921, Z    +0.000, E1    +9.337, E3 +302875.567}
SPL {X  -162.817, Y  +379.558, Z    +0.000, E1    +2.744, E3 +302875.957}
SPL {X  -162.820, Y  +384.383, Z    +0.000, E1    -0.869, E3 +302875.927}
SPL {X  -162.820, Y  +388.871, Z    +0.000, E1    -5.151, E3 +302875.633}
SPL {X  -162.820, Y  +395.861, Z    +0.000, E1   -13.028, E3 +302875.744}
SPL {X  -162.820, Y  +409.049, Z    +0.000, E1   -29.128, E3 +302874.587}
SPL {X  -162.820, Y  +444.592, Z    +0.000, E1   -49.032, E3 +302893.596}
SPL {X  -162.820, Y  +458.217, Z    +0.000, E1   -51.268, E3 +302905.541}
SPL {X  -162.820, Y  +501.848, Z    +0.000, E1   -54.235, E3 +302951.909}
ENDSPLINE

SPLINE
SPL {X  -162.820, Y  +498.156, Z    +0.000, E1   -50.986, E3 +302965.459}
ENDSPLINE

SPLINE
SPL {X  -162.820, Y  +499.429, Z    +0.000, E1   -49.453, E3 +302976.817}
SPL {X  -162.820, Y  +505.173, Z    +0.000, E1   -49.386, E3 +302987.473}
SPL {X  -162.820, Y  +510.642, Z    +0.000, E1   -49.447, E3 +302996.823}
SPL {X  -162.820, Y  +516.435, Z    +0.000, E1   -49.526, E3 +303006.701}
SPL {X  -162.820, Y  +523.383, Z    +0.000, E1   -49.407, E3 +303019.888}
SPL {X  -162.820, Y  +532.283, Z    +0.000, E1   -49.462, E3 +303035.490}
SPL {X  -162.820, Y  +541.471, Z    +0.000, E1   -49.456, E3 +303051.868}
SPL {X  -162.820, Y  +548.933, Z    +0.000, E1   -49.456, E3 +303065.057}
SPL {X  -162.820, Y  +553.997, Z    +0.000, E1   -49.325, E3 +303074.860}
SPL {X  -162.820, Y  +562.346, Z    +0.000, E1   -49.498, E3 +303088.923}
SPL {X  -162.820, Y  +570.444, Z    +0.000, E1   -49.421, E3 +303103.670}
SPL {X  -162.820, Y  +577.429, Z    +0.000, E1   -49.474, E3 +303115.784}
SPL {X  -162.820, Y  +585.965, Z    +0.000, E1   -49.447, E3 +303131.358}
SPL {X  -162.820, Y  +594.192, Z    +0.000, E1   -49.325, E3 +303146.601}
SPL {X  -162.820, Y  +600.267, Z    +0.000, E1   -49.443, E3 +303156.689}
SPL {X  -162.820, Y  +606.218, Z    +0.000, E1   -49.464, E3 +303167.236}
SPL {X  -162.820, Y  +612.538, Z    +0.000, E1   -49.488, E3 +303178.287}
SPL {X  -162.820, Y  +617.738, Z    +0.000, E1   -49.301, E3 +303188.723}
SPL {X  -162.820, Y  +624.265, Z    +0.000, E1   -49.443, E3 +303199.519}
SPL {X  -162.820, Y  +632.551, Z    +0.000, E1   -49.478, E3 +303214.288}
SPL {X  -162.820, Y  +641.207, Z    +0.000, E1   -49.420, E3 +303229.931}
SPL {X  -162.820, Y  +648.011, Z    +0.000, E1   -49.484, E3 +303241.608}
SPL {X  -162.820, Y  +655.976, Z    +0.000, E1   -49.445, E3 +303256.237}
SPL {X  -162.820, Y  +663.916, Z    +0.000, E1   -49.371, E3 +303270.666}
SPL {X  -162.820, Y  +669.755, Z    +0.000, E1   -49.387, E3 +303280.990}
SPL {X  -162.807, Y  +675.597, Z    +0.000, E1   -49.472, E3 +303290.893}
SPL {X  -162.632, Y  +681.322, Z    +0.000, E1   -49.345, E3 +303301.904}
SPL {X  -162.228, Y  +687.372, Z    +0.000, E1   -49.294, E3 +303312.991}
SPL {X  -161.723, Y  +692.372, Z    +0.000, E1   -49.172, E3 +303322.621}
SPL {X  -161.009, Y  +697.714, Z    +0.000, E1   -49.214, E3 +303331.905}
SPL {X  -160.313, Y  +701.965, Z    +0.000, E1   -48.932, E3 +303341.118}
SPL {X  -159.435, Y  +706.528, Z    +0.000, E1   -48.764, E3 +303350.244}
SPL {X  -157.894, Y  +713.249, Z    +0.000, E1   -48.586, E3 +303363.438}
SPL {X  -156.071, Y  +719.891, Z    +0.000, E1   -48.264, E3 +303376.909}
SPL {X  -154.661, Y  +724.395, Z    +0.000, E1   -47.951, E3 +303386.590}
SPL {X  -153.094, Y  +728.931, Z    +0.000, E1   -47.705, E3 +303396.027}
SPL {X  -151.300, Y  +733.655, Z    +0.000, E1   -47.339, E3 +303406.336}
SPL {X  -145.669, Y  +746.239, Z    +0.000, E1   -50.198, E3 +303413.112}
SPL {X  -135.559, Y  +763.690, Z    +0.000, E1   -44.340, E3 +303499.906}
ENDSPLINE

SPLINE
SPL {X  -153.801, Y  +726.938, Z    +0.000, E1   -29.643, E3 +303568.619}
SPL {X  -160.383, Y  +701.564, Z    +0.000, E1   -18.145, E3 +303576.759}
SPL {X  -162.078, Y  +689.023, Z    +0.000, E1   -11.510, E3 +303576.297}
SPL {X  -162.685, Y  +680.136, Z    +0.000, E1    -6.379, E3 +303576.585}
SPL {X  -162.820, Y  +672.919, Z    +0.000, E1    -1.752, E3 +303576.624}
SPL {X  -162.820, Y  +667.861, Z    +0.000, E1    +2.254, E3 +303576.426}
SPL {X  -162.820, Y  +662.755, Z    +0.000, E1    +7.521, E3 +303576.466}
SPL {X  -162.820, Y  +657.537, Z    +0.000, E1   +13.540, E3 +303576.136}
SPL {X  -162.820, Y  +650.460, Z    +0.000, E1   +22.200, E3 +303575.567}
SPL {X  -162.820, Y  +637.843, Z    +0.000, E1   +35.051, E3 +303577.643}
SPL {X  -162.820, Y  +595.072, Z    +0.000, E1   +53.652, E3 +303598.364}
SPL {X  -162.820, Y  +560.706, Z    +0.000, E1   +50.482, E3 +303659.273}
ENDSPLINE

SPLINE
SPL {X  -162.820, Y  +560.978, Z    +0.000, E1   +48.448, E3 +303671.358}
ENDSPLINE

SPLINE
SPL {X  -162.820, Y  +552.125, Z    +0.000, E1   +48.477, E3 +303687.463}
SPL {X  -162.820, Y  +545.800, Z    +0.000, E1   +48.334, E3 +303699.905}
SPL {X  -162.820, Y  +538.900, Z    +0.000, E1   +48.334, E3 +303712.820}
SPL {X  -162.820, Y  +530.572, Z    +0.000, E1   +48.392, E3 +303727.870}
SPL {X  -162.820, Y  +522.157, Z    +0.000, E1   +48.326, E3 +303743.959}
SPL {X  -162.820, Y  +512.600, Z    +0.000, E1   +48.469, E3 +303760.735}
SPL {X  -162.820, Y  +504.728, Z    +0.000, E1   +48.342, E3 +303776.064}
ENDSPLINE

SPLINE
SPL {X  -162.820, Y  +517.326, Z    +0.000, E1   +41.232, E3 +303791.783}
ENDSPLINE

SPLINE
SPL {X  -162.820, Y  +509.871, Z    +0.000, E1   +42.115, E3 +303803.885}
SPL {X  -162.820, Y  +501.934, Z    +0.000, E1   +43.022, E3 +303816.612}
SPL {X  -162.820, Y  +494.356, Z    +0.000, E1   +43.819, E3 +303828.453}
SPL {X  -162.820, Y  +487.058, Z    +0.000, E1   +44.544, E3 +303839.917}
SPL {X  -162.820, Y  +476.193, Z    +0.000, E1   +45.591, E3 +303856.356}
SPL {X  -162.820, Y  +465.836, Z    +0.000, E1   +46.727, E3 +303870.272}
SPL {X  -162.820, Y  +457.217, Z    +0.000, E1   +47.671, E3 +303881.310}
SPL {X  -162.820, Y  +446.677, Z    +0.000, E1   +48.707, E3 +303894.839}
SPL {X  -162.820, Y  +435.978, Z    +0.000, E1   +49.560, E3 +303908.989}
SPL {X  -162.820, Y  +428.488, Z    +0.000, E1   +49.830, E3 +303920.568}
SPL {X  -162.820, Y  +423.062, Z    +0.000, E1   +49.728, E3 +303930.711}
SPL {X  -162.820, Y  +416.560, Z    +0.000, E1   +49.816, E3 +303941.692}
SPL {X  -162.820, Y  +407.996, Z    +0.000, E1   +49.793, E3 +303957.058}
SPL {X  -162.820, Y  +398.766, Z    +0.000, E1   +49.793, E3 +303973.237}
SPL {X  -162.820, Y  +391.831, Z    +0.000, E1   +49.801, E3 +303985.283}
SPL {X  -162.820, Y  +386.334, Z    +0.000, E1   +49.739, E3 +303995.371}
SPL {X  -162.801, Y  +377.981, Z    +0.000, E1   +49.798, E3 +304009.893}
SPL {X  -162.314, Y  +367.677, Z    +0.000, E1   +49.734, E3 +304028.533}
SPL {X  -161.614, Y  +360.718, Z    +0.000, E1   +49.491, E3 +304041.950}
SPL {X  -160.828, Y  +355.106, Z    +0.000, E1   +49.536, E3 +304051.634}
SPL {X  -159.832, Y  +349.452, Z    +0.000, E1   +49.188, E3 +304063.606}
SPL {X  -158.863, Y  +344.823, Z    +0.000, E1   +49.020, E3 +304072.655}
SPL {X  -157.695, Y  +339.971, Z    +0.000, E1   +48.934, E3 +304081.751}
SPL {X  -156.136, Y  +334.326, Z    +0.000, E1   +48.578, E3 +304093.717}
SPL {X  -154.561, Y  +329.302, Z    +0.000, E1   +48.290, E3 +304104.048}
SPL {X  -152.787, Y  +324.229, Z    +0.000, E1   +47.981, E3 +304114.738}
SPL {X  -150.789, Y  +319.074, Z    +0.000, E1   +47.585, E3 +304125.760}
SPL {X  -145.123, Y  +306.679, Z    +0.000, E1   +50.518, E3 +304131.658}
SPL {X  -135.207, Y  +289.783, Z    +0.000, E1   +44.101, E3 +304225.172}
ENDSPLINE

SPLINE
SPL {X  -154.528, Y  +329.203, Z    +0.000, E1   +28.834, E3 +304295.533}
SPL {X  -160.380, Y  +352.419, Z    +0.000, E1   +18.163, E3 +304299.894}
SPL {X  -162.149, Y  +365.734, Z    +0.000, E1   +11.090, E3 +304298.502}
SPL {X  -162.754, Y  +375.862, Z    +0.000, E1    +5.134, E3 +304299.339}
SPL {X  -162.820, Y  +382.085, Z    +0.000, E1    +0.928, E3 +304299.028}
SPL {X  -162.820, Y  +385.149, Z    +0.000, E1    -1.602, E3 +304298.754}
SPL {X  -162.820, Y  +388.871, Z    +0.000, E1    -5.151, E3 +304298.710}
SPL {X  -162.820, Y  +395.861, Z    +0.000, E1   -13.028, E3 +304298.821}
SPL {X  -162.820, Y  +409.049, Z    +0.000, E1   -29.128, E3 +304297.663}
SPL {X  -162.820, Y  +446.299, Z    +0.000, E1   -49.360, E3 +304318.167}
SPL {X  -162.820, Y  +502.427, Z    +0.000, E1   -53.345, E3 +304381.152}
ENDSPLINE

SPLINE
SPL {X  -162.820, Y  +494.458, Z    +0.000, E1   -49.332, E3 +304391.685}
ENDSPLINE

SPLINE
SPL {X  -162.820, Y  +499.429, Z    +0.000, E1   -49.453, E3 +304399.894}
SPL {X  -162.820, Y  +505.173, Z    +0.000, E1   -49.386, E3 +304410.550}
SPL {X  -162.820, Y  +510.642, Z    +0.000, E1   -49.447, E3 +304419.900}
SPL {X  -162.820, Y  +516.435, Z    +0.000, E1   -49.526, E3 +304429.778}
SPL {X  -162.820, Y  +523.383, Z    +0.000, E1   -49.407, E3 +304442.965}
SPL {X  -162.820, Y  +530.598, Z    +0.000, E1   -49.471, E3 +304455.366}
SPL {X  -162.820, Y  +536.932, Z    +0.000, E1   -49.395, E3 +304467.124}
SPL {X  -162.820, Y  +543.021, Z    +0.000, E1   -49.432, E3 +304477.730}
SPL {X  -162.820, Y  +548.933, Z    +0.000, E1   -49.456, E3 +304488.134}
SPL {X  -162.820, Y  +553.997, Z    +0.000, E1   -49.325, E3 +304497.937}
SPL {X  -162.820, Y  +560.268, Z    +0.000, E1   -49.531, E3 +304507.895}
SPL {X  -162.820, Y  +564.590, Z    +0.000, E1   -49.361, E3 +304516.595}
SPL {X  -162.820, Y  +570.444, Z    +0.000, E1   -49.421, E3 +304526.747}
SPL {X  -162.820, Y  +577.429, Z    +0.000, E1   -49.474, E3 +304538.861}
SPL {X  -162.820, Y  +585.965, Z    +0.000, E1   -49.447, E3 +304554.435}
SPL {X  -162.820, Y  +594.192, Z    +0.000, E1   -49.325, E3 +304569.678}
SPL {X  -162.820, Y  +600.267, Z    +0.000, E1   -49.443, E3 +304579.766}
SPL {X  -162.820, Y  +606.218, Z    +0.000, E1   -49.464, E3 +304590.313}
SPL {X  -162.820, Y  +612.538, Z    +0.000, E1   -49.488, E3 +304601.364}
SPL {X  -162.820, Y  +617.738, Z    +0.000, E1   -49.301, E3 +304611.800}
SPL {X  -162.820, Y  +624.265, Z    +0.000, E1   -49.443, E3 +304622.596}
SPL {X  -162.820, Y  +632.551, Z    +0.000, E1   -49.478, E3 +304637.364}
SPL {X  -162.820, Y  +641.207, Z    +0.000, E1   -49.420, E3 +304653.008}
SPL {X  -162.820, Y  +649.864, Z    +0.000, E1   -49.433, E3 +304668.486}
SPL {X  -162.820, Y  +658.147, Z    +0.000, E1   -49.491, E3 +304682.753}
SPL {X  -162.820, Y  +663.916, Z    +0.000, E1   -49.371, E3 +304693.743}
SPL {X  -162.820, Y  +669.755, Z    +0.000, E1   -49.387, E3 +304704.067}
SPL {X  -162.807, Y  +675.597, Z    +0.000, E1   -49.472, E3 +304713.970}
SPL {X  -162.632, Y  +681.322, Z    +0.000, E1   -49.345, E3 +304724.981}
SPL {X  -162.228, Y  +687.372, Z    +0.000, E1   -49.294, E3 +304736.068}
SPL {X  -161.723, Y  +692.372, Z    +0.000, E1   -49.172, E3 +304745.698}
SPL {X  -161.009, Y  +697.714, Z    +0.000, E1   -49.214, E3 +304754.982}
SPL {X  -160.313, Y  +701.965, Z    +0.000, E1   -48.932, E3 +304764.194}
SPL {X  -158.980, Y  +708.651, Z    +0.000, E1   -48.774, E3 +304777.235}
SPL {X  -157.477, Y  +714.869, Z    +0.000, E1   -48.424, E3 +304790.109}
SPL {X  -156.071, Y  +719.891, Z    +0.000, E1   -48.264, E3 +304799.986}
SPL {X  -154.661, Y  +724.395, Z    +0.000, E1   -47.951, E3 +304809.667}
SPL {X  -153.094, Y  +728.931, Z    +0.000, E1   -47.705, E3 +304819.104}
SPL {X  -150.266, Y  +736.194, Z    +0.000, E1   -47.943, E3 +304830.713}
SPL {X  -143.458, Y  +750.508, Z    +0.000, E1   -51.034, E3 +304838.738}
SPL {X  -135.559, Y  +763.690, Z    +0.000, E1   -44.340, E3 +304922.983}
ENDSPLINE

SPLINE
SPL {X  -153.801, Y  +726.938, Z    +0.000, E1   -29.643, E3 +304991.696}
SPL {X  -160.383, Y  +701.564, Z    +0.000, E1   -18.145, E3 +304999.836}
SPL {X  -162.078, Y  +689.023, Z    +0.000, E1   -11.510, E3 +304999.374}
SPL {X  -162.685, Y  +680.136, Z    +0.000, E1    -6.379, E3 +304999.662}
SPL {X  -162.820, Y  +672.919, Z    +0.000, E1    -1.752, E3 +304999.701}
SPL {X  -162.820, Y  +667.861, Z    +0.000, E1    +2.254, E3 +304999.503}
SPL {X  -162.820, Y  +662.755, Z    +0.000, E1    +7.521, E3 +304999.543}
SPL {X  -162.820, Y  +657.537, Z    +0.000, E1   +13.540, E3 +304999.212}
SPL {X  -162.820, Y  +650.460, Z    +0.000, E1   +22.200, E3 +304998.643}
SPL {X  -162.820, Y  +637.843, Z    +0.000, E1   +35.051, E3 +305000.720}
SPL {X  -162.820, Y  +595.072, Z    +0.000, E1   +53.652, E3 +305021.440}
SPL {X  -162.820, Y  +561.831, Z    +0.000, E1   +49.171, E3 +305088.663}
SPL {X  -162.820, Y  +553.813, Z    +0.000, E1   +48.452, E3 +305107.728}
SPL {X  -162.820, Y  +543.226, Z    +0.000, E1   +48.398, E3 +305127.580}
SPL {X  -162.820, Y  +534.689, Z    +0.000, E1   +48.295, E3 +305143.881}
SPL {X  -162.820, Y  +528.564, Z    +0.000, E1   +48.407, E3 +305154.455}
SPL {X  -162.820, Y  +522.157, Z    +0.000, E1   +48.326, E3 +305167.036}
SPL {X  -162.820, Y  +513.750, Z    +0.000, E1   +48.520, E3 +305181.268}
SPL {X  -162.820, Y  +508.282, Z    +0.000, E1   +48.307, E3 +305192.670}
SPL {X  -162.820, Y  +502.890, Z    +0.000, E1   +48.309, E3 +305202.596}
ENDSPLINE

SPLINE
SPL {X  -162.820, Y  +520.386, Z    +0.000, E1   +40.911, E3 +305209.326}
ENDSPLINE

SPLINE
SPL {X  -162.820, Y  +515.876, Z    +0.000, E1   +41.348, E3 +305217.524}
SPL {X  -162.820, Y  +507.007, Z    +0.000, E1   +42.470, E3 +305231.539}
SPL {X  -162.820, Y  +496.780, Z    +0.000, E1   +43.573, E3 +305247.793}
SPL {X  -162.820, Y  +488.962, Z    +0.000, E1   +44.342, E3 +305260.061}
SPL {X  -162.820, Y  +481.373, Z    +0.000, E1   +45.107, E3 +305271.545}
SPL {X  -162.820, Y  +473.909, Z    +0.000, E1   +45.743, E3 +305283.058}
SPL {X  -162.820, Y  +463.464, Z    +0.000, E1   +47.025, E3 +305296.275}
SPL {X  -162.820, Y  +451.336, Z    +0.000, E1   +48.248, E3 +305312.045}
SPL {X  -162.820, Y  +443.046, Z    +0.000, E1   +49.021, E3 +305322.544}
SPL {X  -162.820, Y  +435.978, Z    +0.000, E1   +49.560, E3 +305332.066}
SPL {X  -162.820, Y  +428.488, Z    +0.000, E1   +49.830, E3 +305343.645}
SPL {X  -162.820, Y  +423.062, Z    +0.000, E1   +49.728, E3 +305353.788}
SPL {X  -162.820, Y  +416.560, Z    +0.000, E1   +49.816, E3 +305364.769}
SPL {X  -162.820, Y  +407.996, Z    +0.000, E1   +49.793, E3 +305380.135}
SPL {X  -162.820, Y  +400.367, Z    +0.000, E1   +49.822, E3 +305393.193}
SPL {X  -162.820, Y  +393.582, Z    +0.000, E1   +49.779, E3 +305405.511}
SPL {X  -162.820, Y  +384.205, Z    +0.000, E1   +49.756, E3 +305422.291}
SPL {X  -162.753, Y  +375.844, Z    +0.000, E1   +49.816, E3 +305436.467}
SPL {X  -162.415, Y  +369.029, Z    +0.000, E1   +49.751, E3 +305448.956}
SPL {X  -161.760, Y  +361.947, Z    +0.000, E1   +49.515, E3 +305462.795}
SPL {X  -160.828, Y  +355.106, Z    +0.000, E1   +49.536, E3 +305474.711}
SPL {X  -159.832, Y  +349.452, Z    +0.000, E1   +49.188, E3 +305486.682}
SPL {X  -158.863, Y  +344.823, Z    +0.000, E1   +49.020, E3 +305495.732}
SPL {X  -157.695, Y  +339.971, Z    +0.000, E1   +48.934, E3 +305504.828}
SPL {X  -156.136, Y  +334.326, Z    +0.000, E1   +48.578, E3 +305516.794}
SPL {X  -154.561, Y  +329.302, Z    +0.000, E1   +48.290, E3 +305527.125}
SPL {X  -152.787, Y  +324.229, Z    +0.000, E1   +47.981, E3 +305537.815}
SPL {X  -150.789, Y  +319.074, Z    +0.000, E1   +47.585, E3 +305548.837}
SPL {X  -145.123, Y  +306.679, Z    +0.000, E1   +50.518, E3 +305554.735}
SPL {X  -135.207, Y  +289.783, Z    +0.000, E1   +44.101, E3 +305648.249}
ENDSPLINE

SPLINE
SPL {X  -154.528, Y  +329.203, Z    +0.000, E1   +28.834, E3 +305718.610}
SPL {X  -160.380, Y  +352.419, Z    +0.000, E1   +18.163, E3 +305722.971}
SPL {X  -162.408, Y  +368.921, Z    +0.000, E1    +9.337, E3 +305721.721}
SPL {X  -162.817, Y  +379.558, Z    +0.000, E1    +2.744, E3 +305722.111}
SPL {X  -162.820, Y  +383.077, Z    +0.000, E1    +0.110, E3 +305722.506}
SPL {X  -162.820, Y  +386.028, Z    +0.000, E1    -2.328, E3 +305721.829}
SPL {X  -162.820, Y  +389.792, Z    +0.000, E1    -6.211, E3 +305721.761}
SPL {X  -162.820, Y  +395.861, Z    +0.000, E1   -13.028, E3 +305721.898}
SPL {X  -162.820, Y  +409.049, Z    +0.000, E1   -29.128, E3 +305720.740}
SPL {X  -162.820, Y  +446.299, Z    +0.000, E1   -49.360, E3 +305741.244}
SPL {X  -162.820, Y  +502.427, Z    +0.000, E1   -53.345, E3 +305804.229}
ENDSPLINE

SPLINE
SPL {X  -162.820, Y  +494.458, Z    +0.000, E1   -49.332, E3 +305814.761}
ENDSPLINE

SPLINE
SPL {X  -162.820, Y  +499.429, Z    +0.000, E1   -49.453, E3 +305822.971}
SPL {X  -162.820, Y  +505.173, Z    +0.000, E1   -49.386, E3 +305833.626}
SPL {X  -162.820, Y  +510.642, Z    +0.000, E1   -49.447, E3 +305842.977}
SPL {X  -162.820, Y  +516.435, Z    +0.000, E1   -49.526, E3 +305852.855}
SPL {X  -162.820, Y  +522.095, Z    +0.000, E1   -49.420, E3 +305863.551}
SPL {X  -162.820, Y  +529.397, Z    +0.000, E1   -49.440, E3 +305876.560}
SPL {X  -162.820, Y  +536.932, Z    +0.000, E1   -49.395, E3 +305890.201}
SPL {X  -162.820, Y  +543.021, Z    +0.000, E1   -49.432, E3 +305900.807}
SPL {X  -162.820, Y  +548.933, Z    +0.000, E1   -49.456, E3 +305911.210}
SPL {X  -162.820, Y  +553.997, Z    +0.000, E1   -49.325, E3 +305921.014}
SPL {X  -162.820, Y  +562.346, Z    +0.000, E1   -49.498, E3 +305935.077}
SPL {X  -162.820, Y  +570.444, Z    +0.000, E1   -49.421, E3 +305949.823}
SPL {X  -162.820, Y  +577.429, Z    +0.000, E1   -49.474, E3 +305961.938}
SPL {X  -162.820, Y  +585.965, Z    +0.000, E1   -49.447, E3 +305977.512}
SPL {X  -162.820, Y  +594.192, Z    +0.000, E1   -49.325, E3 +305992.755}
SPL {X  -162.820, Y  +600.267, Z    +0.000, E1   -49.443, E3 +306002.843}
SPL {X  -162.820, Y  +606.218, Z    +0.000, E1   -49.464, E3 +306013.390}
SPL {X  -162.820, Y  +612.538, Z    +0.000, E1   -49.488, E3 +306024.441}
SPL {X  -162.820, Y  +617.738, Z    +0.000, E1   -49.301, E3 +306034.877}
SPL {X  -162.820, Y  +624.265, Z    +0.000, E1   -49.443, E3 +306045.673}
SPL {X  -162.820, Y  +632.551, Z    +0.000, E1   -49.478, E3 +306060.441}
SPL {X  -162.820, Y  +641.207, Z    +0.000, E1   -49.420, E3 +306076.085}
SPL {X  -162.820, Y  +649.864, Z    +0.000, E1   -49.433, E3 +306091.563}
SPL {X  -162.820, Y  +658.147, Z    +0.000, E1   -49.491, E3 +306105.830}
SPL {X  -162.820, Y  +663.916, Z    +0.000, E1   -49.371, E3 +306116.819}
SPL {X  -162.820, Y  +669.755, Z    +0.000, E1   -49.387, E3 +306127.144}
SPL {X  -162.807, Y  +675.597, Z    +0.000, E1   -49.472, E3 +306137.047}
SPL {X  -162.632, Y  +681.322, Z    +0.000, E1   -49.345, E3 +306148.058}
SPL {X  -162.228, Y  +687.372, Z    +0.000, E1   -49.294, E3 +306159.145}
SPL {X  -161.723, Y  +692.372, Z    +0.000, E1   -49.172, E3 +306168.775}
SPL {X  -161.009, Y  +697.714, Z    +0.000, E1   -49.214, E3 +306178.059}
SPL {X  -160.313, Y  +701.965, Z    +0.000, E1   -48.932, E3 +306187.271}
SPL {X  -158.980, Y  +708.651, Z    +0.000, E1   -48.774, E3 +306200.312}
SPL {X  -157.477, Y  +714.869, Z    +0.000, E1   -48.424, E3 +306213.186}
SPL {X  -156.071, Y  +719.891, Z    +0.000, E1   -48.264, E3 +306223.063}
SPL {X  -154.661, Y  +724.395, Z    +0.000, E1   -47.951, E3 +306232.744}
SPL {X  -153.094, Y  +728.931, Z    +0.000, E1   -47.705, E3 +306242.181}
SPL {X  -151.300, Y  +733.655, Z    +0.000, E1   -47.339, E3 +306252.489}
SPL {X  -145.669, Y  +746.239, Z    +0.000, E1   -50.198, E3 +306259.266}
SPL {X  -135.084, Y  +764.399, Z    +0.000, E1   -44.787, E3 +306342.170}
ENDSPLINE

SPLINE
SPL {X  -153.038, Y  +729.086, Z    +0.000, E1   -30.522, E3 +306412.877}
SPL {X  -160.383, Y  +701.564, Z    +0.000, E1   -18.145, E3 +306422.913}
SPL {X  -162.078, Y  +689.023, Z    +0.000, E1   -11.510, E3 +306422.451}
SPL {X  -162.685, Y  +680.136, Z    +0.000, E1    -6.379, E3 +306422.739}
SPL {X  -162.820, Y  +672.919, Z    +0.000, E1    -1.752, E3 +306422.778}
SPL {X  -162.820, Y  +667.861, Z    +0.000, E1    +2.254, E3 +306422.579}
SPL {X  -162.820, Y  +662.755, Z    +0.000, E1    +7.521, E3 +306422.620}
SPL {X  -162.820, Y  +657.537, Z    +0.000, E1   +13.540, E3 +306422.289}
SPL {X  -162.820, Y  +650.460, Z    +0.000, E1   +22.200, E3 +306421.720}
SPL {X  -162.820, Y  +637.843, Z    +0.000, E1   +35.051, E3 +306423.797}
SPL {X  -162.820, Y  +595.072, Z    +0.000, E1   +53.652, E3 +306444.517}
SPL {X  -162.820, Y  +561.831, Z    +0.000, E1   +49.171, E3 +306511.740}
SPL {X  -162.820, Y  +555.289, Z    +0.000, E1   +48.406, E3 +306528.201}
SPL {X  -162.820, Y  +547.003, Z    +0.000, E1   +48.390, E3 +306543.613}
SPL {X  -162.820, Y  +540.645, Z    +0.000, E1   +48.364, E3 +306555.409}
SPL {X  -162.820, Y  +534.689, Z    +0.000, E1   +48.295, E3 +306566.958}
SPL {X  -162.820, Y  +528.564, Z    +0.000, E1   +48.407, E3 +306577.531}
SPL {X  -162.820, Y  +522.157, Z    +0.000, E1   +48.326, E3 +306590.113}
SPL {X  -162.820, Y  +513.750, Z    +0.000, E1   +48.520, E3 +306604.344}
SPL {X  -162.820, Y  +508.282, Z    +0.000, E1   +48.307, E3 +306615.747}
SPL {X  -162.820, Y  +502.890, Z    +0.000, E1   +48.309, E3 +306625.673}
ENDSPLINE

SPLINE
SPL {X  -162.820, Y  +517.326, Z    +0.000, E1   +41.232, E3 +306637.937}
ENDSPLINE

SPLINE
SPL {X  -162.820, Y  +509.871, Z    +0.000, E1   +42.115, E3 +306650.039}
SPL {X  -162.820, Y  +501.934, Z    +0.000, E1   +43.022, E3 +306662.765}
SPL {X  -162.820, Y  +494.356, Z    +0.000, E1   +43.819, E3 +306674.607}
SPL {X  -162.820, Y  +487.058, Z    +0.000, E1   +44.544, E3 +306686.071}
SPL {X  -162.820, Y  +476.193, Z    +0.000, E1   +45.591, E3 +306702.510}
SPL {X  -162.820, Y  +465.836, Z    +0.000, E1   +46.727, E3 +306716.426}
SPL {X  -162.820, Y  +457.217, Z    +0.000, E1   +47.671, E3 +306727.464}
SPL {X  -162.820, Y  +449.104, Z    +0.000, E1   +48.459, E3 +306737.932}
SPL {X  -162.820, Y  +438.072, Z    +0.000, E1   +49.432, E3 +306752.287}
SPL {X  -162.820, Y  +428.488, Z    +0.000, E1   +49.830, E3 +306766.722}
SPL {X  -162.820, Y  +423.062, Z    +0.000, E1   +49.728, E3 +306776.865}
SPL {X  -162.820, Y  +416.560, Z    +0.000, E1   +49.816, E3 +306787.846}
SPL {X  -162.820, Y  +410.559, Z    +0.000, E1   +49.727, E3 +306798.901}
SPL {X  -162.820, Y  +405.170, Z    +0.000, E1   +49.772, E3 +306808.103}
SPL {X  -162.820, Y  +398.766, Z    +0.000, E1   +49.793, E3 +306819.391}
SPL {X  -162.820, Y  +391.831, Z    +0.000, E1   +49.801, E3 +306831.437}
SPL {X  -162.820, Y  +386.334, Z    +0.000, E1   +49.739, E3 +306841.525}
SPL {X  -162.801, Y  +377.981, Z    +0.000, E1   +49.798, E3 +306856.047}
SPL {X  -162.314, Y  +367.677, Z    +0.000, E1   +49.734, E3 +306874.686}
SPL {X  -161.359, Y  +358.734, Z    +0.000, E1   +49.535, E3 +306891.470}
SPL {X  -160.051, Y  +350.597, Z    +0.000, E1   +49.332, E3 +306907.080}
SPL {X  -158.863, Y  +344.823, Z    +0.000, E1   +49.020, E3 +306918.808}
SPL {X  -157.695, Y  +339.971, Z    +0.000, E1   +48.934, E3 +306927.905}
SPL {X  -156.136, Y  +334.326, Z    +0.000, E1   +48.578, E3 +306939.871}
SPL {X  -154.561, Y  +329.302, Z    +0.000, E1   +48.290, E3 +306950.202}
SPL {X  -152.787, Y  +324.229, Z    +0.000, E1   +47.981, E3 +306960.892}
SPL {X  -150.789, Y  +319.074, Z    +0.000, E1   +47.585, E3 +306971.914}
SPL {X  -145.123, Y  +306.679, Z    +0.000, E1   +50.518, E3 +306977.812}
SPL {X  -135.207, Y  +289.783, Z    +0.000, E1   +44.101, E3 +307071.326}
ENDSPLINE

SPLINE
SPL {X  -154.528, Y  +329.203, Z    +0.000, E1   +28.834, E3 +307141.687}
SPL {X  -160.380, Y  +352.419, Z    +0.000, E1   +18.163, E3 +307146.048}
SPL {X  -162.149, Y  +365.734, Z    +0.000, E1   +11.090, E3 +307144.656}
SPL {X  -162.754, Y  +375.862, Z    +0.000, E1    +5.134, E3 +307145.493}
SPL {X  -162.820, Y  +382.085, Z    +0.000, E1    +0.928, E3 +307145.182}
SPL {X  -162.820, Y  +386.028, Z    +0.000, E1    -2.328, E3 +307144.906}
SPL {X  -162.820, Y  +389.792, Z    +0.000, E1    -6.211, E3 +307144.838}
SPL {X  -162.820, Y  +394.068, Z    +0.000, E1   -11.043, E3 +307144.955}
SPL {X  -162.820, Y  +398.921, Z    +0.000, E1   -16.945, E3 +307145.008}
SPL {X  -162.820, Y  +409.049, Z    +0.000, E1   -29.128, E3 +307143.817}
SPL {X  -162.820, Y  +446.299, Z    +0.000, E1   -49.360, E3 +307164.321}
SPL {X  -162.820, Y  +502.427, Z    +0.000, E1   -53.345, E3 +307227.306}
ENDSPLINE

SPLINE
SPL {X  -162.820, Y  +497.758, Z    +0.000, E1   -49.444, E3 +307243.245}
ENDSPLINE

SPLINE
SPL {X  -162.820, Y  +507.703, Z    +0.000, E1   -49.462, E3 +307260.963}
SPL {X  -162.820, Y  +516.435, Z    +0.000, E1   -49.526, E3 +307275.931}
SPL {X  -162.820, Y  +522.095, Z    +0.000, E1   -49.420, E3 +307286.628}
SPL {X  -162.820, Y  +529.397, Z    +0.000, E1   -49.440, E3 +307299.637}
SPL {X  -162.820, Y  +536.932, Z    +0.000, E1   -49.395, E3 +307313.278}
SPL {X  -162.820, Y  +543.021, Z    +0.000, E1   -49.432, E3 +307323.884}
SPL {X  -162.820, Y  +548.933, Z    +0.000, E1   -49.456, E3 +307334.287}
SPL {X  -162.820, Y  +553.997, Z    +0.000, E1   -49.325, E3 +307344.091}
SPL {X  -162.820, Y  +562.346, Z    +0.000, E1   -49.498, E3 +307358.154}
SPL {X  -162.820, Y  +570.444, Z    +0.000, E1   -49.421, E3 +307372.900}
SPL {X  -162.820, Y  +577.429, Z    +0.000, E1   -49.474, E3 +307385.015}
SPL {X  -162.820, Y  +582.387, Z    +0.000, E1   -49.269, E3 +307395.036}
SPL {X  -162.820, Y  +588.456, Z    +0.000, E1   -49.496, E3 +307404.550}
SPL {X  -162.820, Y  +594.192, Z    +0.000, E1   -49.325, E3 +307415.832}
SPL {X  -162.820, Y  +600.267, Z    +0.000, E1   -49.443, E3 +307425.920}
SPL {X  -162.820, Y  +606.218, Z    +0.000, E1   -49.464, E3 +307436.467}
SPL {X  -162.820, Y  +612.538, Z    +0.000, E1   -49.488, E3 +307447.518}
SPL {X  -162.820, Y  +617.738, Z    +0.000, E1   -49.301, E3 +307457.954}
SPL {X  -162.820, Y  +624.265, Z    +0.000, E1   -49.443, E3 +307468.750}
SPL {X  -162.820, Y  +632.551, Z    +0.000, E1   -49.478, E3 +307483.518}
SPL {X  -162.820, Y  +641.207, Z    +0.000, E1   -49.420, E3 +307499.162}
SPL {X  -162.820, Y  +648.011, Z    +0.000, E1   -49.484, E3 +307510.839}
SPL {X  -162.820, Y  +655.976, Z    +0.000, E1   -49.445, E3 +307525.467}
SPL {X  -162.820, Y  +663.916, Z    +0.000, E1   -49.371, E3 +307539.896}
SPL {X  -162.820, Y  +669.755, Z    +0.000, E1   -49.387, E3 +307550.221}
SPL {X  -162.807, Y  +675.597, Z    +0.000, E1   -49.472, E3 +307560.124}
SPL {X  -162.632, Y  +681.322, Z    +0.000, E1   -49.345, E3 +307571.135}
SPL {X  -162.228, Y  +687.372, Z    +0.000, E1   -49.294, E3 +307582.221}
SPL {X  -161.723, Y  +692.372, Z    +0.000, E1   -49.172, E3 +307591.852}
SPL {X  -161.009, Y  +697.714, Z    +0.000, E1   -49.214, E3 +307601.136}
SPL {X  -160.313, Y  +701.965, Z    +0.000, E1   -48.932, E3 +307610.348}
SPL {X  -159.435, Y  +706.528, Z    +0.000, E1   -48.764, E3 +307619.475}
SPL {X  -157.894, Y  +713.249, Z    +0.000, E1   -48.586, E3 +307632.669}
SPL {X  -156.071, Y  +719.891, Z    +0.000, E1   -48.264, E3 +307646.140}
SPL {X  -154.661, Y  +724.395, Z    +0.000, E1   -47.951, E3 +307655.821}
SPL {X  -153.094, Y  +728.931, Z    +0.000, E1   -47.705, E3 +307665.258}
SPL {X  -151.300, Y  +733.655, Z    +0.000, E1   -47.339, E3 +307675.566}
SPL {X  -145.669, Y  +746.239, Z    +0.000, E1   -50.198, E3 +307682.343}
SPL {X  -135.084, Y  +764.399, Z    +0.000, E1   -44.787, E3 +307765.247}
ENDSPLINE

SPLINE
SPL {X  -153.038, Y  +729.086, Z    +0.000, E1   -30.522, E3 +307835.953}
SPL {X  -160.383, Y  +701.564, Z    +0.000, E1   -18.145, E3 +307845.990}
SPL {X  -162.078, Y  +689.023, Z    +0.000, E1   -11.510, E3 +307845.528}
SPL {X  -162.685, Y  +680.136, Z    +0.000, E1    -6.379, E3 +307845.816}
SPL {X  -162.820, Y  +672.919, Z    +0.000, E1    -1.752, E3 +307845.855}
SPL {X  -162.820, Y  +669.270, Z    +0.000, E1    +1.140, E3 +307845.338}
SPL {X  -162.820, Y  +666.754, Z    +0.000, E1    +3.396, E3 +307845.907}
SPL {X  -162.820, Y  +662.755, Z    +0.000, E1    +7.521, E3 +307845.697}
SPL {X  -162.820, Y  +657.537, Z    +0.000, E1   +13.540, E3 +307845.366}
SPL {X  -162.820, Y  +650.460, Z    +0.000, E1   +22.200, E3 +307844.797}
SPL {X  -162.820, Y  +637.843, Z    +0.000, E1   +35.051, E3 +307846.874}
SPL {X  -162.820, Y  +595.072, Z    +0.000, E1   +53.652, E3 +307867.594}
SPL {X  -162.820, Y  +560.706, Z    +0.000, E1   +50.482, E3 +307928.503}
ENDSPLINE

SPLINE
SPL {X  -162.820, Y  +560.978, Z    +0.000, E1   +48.448, E3 +307940.589}
ENDSPLINE

SPLINE
SPL {X  -162.820, Y  +552.125, Z    +0.000, E1   +48.477, E3 +307956.694}
SPL {X  -162.820, Y  +545.800, Z    +0.000, E1   +48.334, E3 +307969.136}
SPL {X  -162.820, Y  +540.645, Z    +0.000, E1   +48.364, E3 +307978.486}
SPL {X  -162.820, Y  +534.689, Z    +0.000, E1   +48.295, E3 +307990.035}
SPL {X  -162.820, Y  +526.053, Z    +0.000, E1   +48.382, E3 +308005.610}
SPL {X  -162.820, Y  +519.666, Z    +0.000, E1   +48.261, E3 +308017.979}
SPL {X  -162.820, Y  +512.600, Z    +0.000, E1   +48.469, E3 +308029.965}
SPL {X  -162.820, Y  +504.728, Z    +0.000, E1   +48.342, E3 +308045.294}
ENDSPLINE

SPLINE
SPL {X  -162.820, Y  +517.326, Z    +0.000, E1   +41.232, E3 +308061.014}
ENDSPLINE

SPLINE
SPL {X  -162.820, Y  +509.871, Z    +0.000, E1   +42.115, E3 +308073.116}
SPL {X  -162.820, Y  +501.934, Z    +0.000, E1   +43.022, E3 +308085.842}
SPL {X  -162.820, Y  +494.356, Z    +0.000, E1   +43.819, E3 +308097.684}
SPL {X  -162.820, Y  +487.058, Z    +0.000, E1   +44.544, E3 +308109.147}
SPL {X  -162.820, Y  +476.193, Z    +0.000, E1   +45.591, E3 +308125.586}
SPL {X  -162.820, Y  +465.836, Z    +0.000, E1   +46.727, E3 +308139.503}
SPL {X  -162.820, Y  +457.217, Z    +0.000, E1   +47.671, E3 +308150.541}
SPL {X  -162.820, Y  +446.677, Z    +0.000, E1   +48.707, E3 +308164.070}
SPL {X  -162.820, Y  +435.978, Z    +0.000, E1   +49.560, E3 +308178.220}
SPL {X  -162.820, Y  +428.488, Z    +0.000, E1   +49.830, E3 +308189.799}
SPL {X  -162.820, Y  +423.062, Z    +0.000, E1   +49.728, E3 +308199.942}
SPL {X  -162.820, Y  +416.560, Z    +0.000, E1   +49.816, E3 +308210.923}
SPL {X  -162.820, Y  +407.996, Z    +0.000, E1   +49.793, E3 +308226.289}
SPL {X  -162.820, Y  +398.766, Z    +0.000, E1   +49.793, E3 +308242.468}
SPL {X  -162.820, Y  +391.831, Z    +0.000, E1   +49.801, E3 +308254.513}
SPL {X  -162.820, Y  +386.334, Z    +0.000, E1   +49.739, E3 +308264.602}
SPL {X  -162.801, Y  +377.981, Z    +0.000, E1   +49.798, E3 +308279.124}
SPL {X  -162.314, Y  +367.677, Z    +0.000, E1   +49.734, E3 +308297.763}
SPL {X  -161.359, Y  +358.734, Z    +0.000, E1   +49.535, E3 +308314.547}
SPL {X  -160.051, Y  +350.597, Z    +0.000, E1   +49.332, E3 +308330.157}
SPL {X  -158.863, Y  +344.823, Z    +0.000, E1   +49.020, E3 +308341.885}
SPL {X  -157.695, Y  +339.971, Z    +0.000, E1   +48.934, E3 +308350.982}
SPL {X  -156.136, Y  +334.326, Z    +0.000, E1   +48.578, E3 +308362.948}
SPL {X  -153.956, Y  +327.511, Z    +0.000, E1   +48.205, E3 +308377.070}
SPL {X  -151.655, Y  +321.245, Z    +0.000, E1   +47.770, E3 +308390.279}
SPL {X  -148.347, Y  +313.391, Z    +0.000, E1   +48.924, E3 +308397.877}
SPL {X  -143.047, Y  +302.732, Z    +0.000, E1   +51.043, E3 +308404.397}
SPL {X  -135.207, Y  +289.783, Z    +0.000, E1   +44.101, E3 +308494.403}
ENDSPLINE

SPLINE
SPL {X  -154.528, Y  +329.203, Z    +0.000, E1   +28.834, E3 +308564.764}
SPL {X  -160.380, Y  +352.419, Z    +0.000, E1   +18.163, E3 +308569.125}
SPL {X  -162.149, Y  +365.734, Z    +0.000, E1   +11.090, E3 +308567.733}
SPL {X  -162.754, Y  +375.862, Z    +0.000, E1    +5.134, E3 +308568.570}
SPL {X  -162.820, Y  +382.085, Z    +0.000, E1    +0.928, E3 +308568.259}
SPL {X  -162.820, Y  +385.149, Z    +0.000, E1    -1.602, E3 +308567.985}
SPL {X  -162.820, Y  +388.871, Z    +0.000, E1    -5.151, E3 +308567.941}
SPL {X  -162.820, Y  +395.861, Z    +0.000, E1   -13.028, E3 +308568.052}
SPL {X  -162.820, Y  +409.049, Z    +0.000, E1   -29.128, E3 +308566.894}
SPL {X  -162.820, Y  +444.592, Z    +0.000, E1   -49.032, E3 +308585.904}
SPL {X  -162.820, Y  +458.217, Z    +0.000, E1   -51.268, E3 +308597.849}
SPL {X  -162.820, Y  +501.848, Z    +0.000, E1   -54.235, E3 +308644.217}
ENDSPLINE

SPLINE
SPL {X  -162.820, Y  +498.156, Z    +0.000, E1   -50.986, E3 +308657.766}
ENDSPLINE

SPLINE
SPL {X  -162.820, Y  +499.429, Z    +0.000, E1   -49.453, E3 +308669.125}
SPL {X  -162.820, Y  +505.173, Z    +0.000, E1   -49.386, E3 +308679.780}
SPL {X  -162.820, Y  +510.642, Z    +0.000, E1   -49.447, E3 +308689.130}
SPL {X  -162.820, Y  +516.435, Z    +0.000, E1   -49.526, E3 +308699.008}
SPL {X  -162.820, Y  +522.095, Z    +0.000, E1   -49.420, E3 +308709.705}
SPL {X  -162.820, Y  +529.397, Z    +0.000, E1   -49.440, E3 +308722.714}
SPL {X  -162.820, Y  +536.932, Z    +0.000, E1   -49.395, E3 +308736.355}
SPL {X  -162.820, Y  +543.021, Z    +0.000, E1   -49.432, E3 +308746.961}
SPL {X  -162.820, Y  +548.933, Z    +0.000, E1   -49.456, E3 +308757.364}
SPL {X  -162.820, Y  +553.997, Z    +0.000, E1   -49.325, E3 +308767.168}
SPL {X  -162.820, Y  +562.346, Z    +0.000, E1   -49.498, E3 +308781.231}
SPL {X  -162.820, Y  +570.444, Z    +0.000, E1   -49.421, E3 +308795.977}
SPL {X  -162.820, Y  +577.429, Z    +0.000, E1   -49.474, E3 +308808.092}
SPL {X  -162.820, Y  +585.965, Z    +0.000, E1   -49.447, E3 +308823.665}
SPL {X  -162.820, Y  +594.192, Z    +0.000, E1   -49.325, E3 +308838.908}
SPL {X  -162.820, Y  +600.267, Z    +0.000, E1   -49.443, E3 +308848.997}
SPL {X  -162.820, Y  +606.218, Z    +0.000, E1   -49.464, E3 +308859.544}
SPL {X  -162.820, Y  +612.538, Z    +0.000, E1   -49.488, E3 +308870.595}
SPL {X  -162.820, Y  +617.738, Z    +0.000, E1   -49.301, E3 +308881.031}
SPL {X  -162.820, Y  +624.265, Z    +0.000, E1   -49.443, E3 +308891.826}
SPL {X  -162.820, Y  +630.226, Z    +0.000, E1   -49.472, E3 +308902.275}
SPL {X  -162.820, Y  +635.239, Z    +0.000, E1   -49.373, E3 +308911.770}
SPL {X  -162.820, Y  +641.207, Z    +0.000, E1   -49.420, E3 +308922.238}
SPL {X  -162.820, Y  +649.864, Z    +0.000, E1   -49.433, E3 +308937.717}
SPL {X  -162.820, Y  +658.147, Z    +0.000, E1   -49.491, E3 +308951.984}
SPL {X  -162.820, Y  +663.916, Z    +0.000, E1   -49.371, E3 +308962.973}
SPL {X  -162.820, Y  +669.755, Z    +0.000, E1   -49.387, E3 +308973.298}
SPL {X  -162.807, Y  +675.597, Z    +0.000, E1   -49.472, E3 +308983.201}
SPL {X  -162.632, Y  +681.322, Z    +0.000, E1   -49.345, E3 +308994.212}
SPL {X  -162.228, Y  +687.372, Z    +0.000, E1   -49.294, E3 +309005.298}
SPL {X  -161.723, Y  +692.372, Z    +0.000, E1   -49.172, E3 +309014.929}
SPL {X  -161.009, Y  +697.714, Z    +0.000, E1   -49.214, E3 +309024.213}
SPL {X  -160.313, Y  +701.965, Z    +0.000, E1   -48.932, E3 +309033.425}
SPL {X  -158.980, Y  +708.651, Z    +0.000, E1   -48.774, E3 +309046.466}
SPL {X  -157.477, Y  +714.869, Z    +0.000, E1   -48.424, E3 +309059.340}
SPL {X  -156.071, Y  +719.891, Z    +0.000, E1   -48.264, E3 +309069.217}
SPL {X  -154.661, Y  +724.395, Z    +0.000, E1   -47.951, E3 +309078.898}
SPL {X  -153.094, Y  +728.931, Z    +0.000, E1   -47.705, E3 +309088.335}
SPL {X  -151.300, Y  +733.655, Z    +0.000, E1   -47.339, E3 +309098.643}
SPL {X  -145.669, Y  +746.239, Z    +0.000, E1   -50.198, E3 +309105.420}
SPL {X  -135.559, Y  +763.690, Z    +0.000, E1   -44.340, E3 +309192.214}
ENDSPLINE

SPLINE
SPL {X  -153.801, Y  +726.938, Z    +0.000, E1   -29.643, E3 +309260.927}
SPL {X  -160.383, Y  +701.564, Z    +0.000, E1   -18.145, E3 +309269.066}
SPL {X  -162.078, Y  +689.023, Z    +0.000, E1   -11.510, E3 +309268.604}
SPL {X  -162.685, Y  +680.136, Z    +0.000, E1    -6.379, E3 +309268.893}
SPL {X  -162.820, Y  +672.919, Z    +0.000, E1    -1.752, E3 +309268.932}
SPL {X  -162.820, Y  +667.861, Z    +0.000, E1    +2.254, E3 +309268.733}
SPL {X  -162.820, Y  +662.755, Z    +0.000, E1    +7.521, E3 +309268.774}
SPL {X  -162.820, Y  +657.537, Z    +0.000, E1   +13.540, E3 +309268.443}
SPL {X  -162.820, Y  +650.460, Z    +0.000, E1   +22.200, E3 +309267.874}
SPL {X  -162.820, Y  +637.843, Z    +0.000, E1   +35.051, E3 +309269.951}
SPL {X  -162.820, Y  +595.072, Z    +0.000, E1   +53.652, E3 +309290.671}
SPL {X  -162.820, Y  +561.831, Z    +0.000, E1   +49.171, E3 +309357.894}
SPL {X  -162.820, Y  +553.813, Z    +0.000, E1   +48.452, E3 +309376.959}
SPL {X  -162.820, Y  +543.226, Z    +0.000, E1   +48.398, E3 +309396.811}
SPL {X  -162.820, Y  +534.689, Z    +0.000, E1   +48.295, E3 +309413.112}
SPL {X  -162.820, Y  +528.564, Z    +0.000, E1   +48.407, E3 +309423.685}
SPL {X  -162.820, Y  +522.157, Z    +0.000, E1   +48.326, E3 +309436.267}
SPL {X  -162.820, Y  +513.750, Z    +0.000, E1   +48.520, E3 +309450.498}
SPL {X  -162.820, Y  +508.282, Z    +0.000, E1   +48.307, E3 +309461.900}
SPL {X  -162.820, Y  +502.890, Z    +0.000, E1   +48.309, E3 +309471.827}
ENDSPLINE

SPLINE
SPL {X  -162.820, Y  +520.386, Z    +0.000, E1   +40.911, E3 +309478.557}
ENDSPLINE

SPLINE
SPL {X  -162.820, Y  +515.876, Z    +0.000, E1   +41.348, E3 +309486.755}
SPL {X  -162.820, Y  +509.871, Z    +0.000, E1   +42.115, E3 +309496.193}
SPL {X  -162.820, Y  +504.481, Z    +0.000, E1   +42.725, E3 +309504.857}
SPL {X  -162.820, Y  +496.780, Z    +0.000, E1   +43.573, E3 +309517.024}
SPL {X  -162.820, Y  +488.962, Z    +0.000, E1   +44.342, E3 +309529.292}
SPL {X  -162.820, Y  +481.373, Z    +0.000, E1   +45.107, E3 +309540.776}
SPL {X  -162.820, Y  +473.909, Z    +0.000, E1   +45.743, E3 +309552.289}
SPL {X  -162.820, Y  +463.464, Z    +0.000, E1   +47.025, E3 +309565.506}
SPL {X  -162.820, Y  +451.336, Z    +0.000, E1   +48.248, E3 +309581.276}
SPL {X  -162.820, Y  +443.046, Z    +0.000, E1   +49.021, E3 +309591.775}
SPL {X  -162.820, Y  +435.978, Z    +0.000, E1   +49.560, E3 +309601.296}
SPL {X  -162.820, Y  +428.488, Z    +0.000, E1   +49.830, E3 +309612.876}
SPL {X  -162.820, Y  +423.062, Z    +0.000, E1   +49.728, E3 +309623.019}
SPL {X  -162.820, Y  +416.560, Z    +0.000, E1   +49.816, E3 +309634.000}
SPL {X  -162.820, Y  +410.559, Z    +0.000, E1   +49.727, E3 +309645.055}
SPL {X  -162.820, Y  +402.501, Z    +0.000, E1   +49.838, E3 +309658.744}
SPL {X  -162.820, Y  +393.582, Z    +0.000, E1   +49.779, E3 +309674.741}
SPL {X  -162.820, Y  +386.334, Z    +0.000, E1   +49.739, E3 +309687.679}
SPL {X  -162.820, Y  +381.297, Z    +0.000, E1   +49.665, E3 +309696.950}
SPL {X  -162.709, Y  +374.487, Z    +0.000, E1   +49.773, E3 +309708.475}
SPL {X  -162.299, Y  +367.483, Z    +0.000, E1   +49.784, E3 +309720.617}
SPL {X  -161.760, Y  +361.947, Z    +0.000, E1   +49.515, E3 +309732.025}
SPL {X  -160.828, Y  +355.106, Z    +0.000, E1   +49.536, E3 +309743.942}
SPL {X  -159.832, Y  +349.452, Z    +0.000, E1   +49.188, E3 +309755.913}
SPL {X  -158.863, Y  +344.823, Z    +0.000, E1   +49.020, E3 +309764.962}
SPL {X  -157.695, Y  +339.971, Z    +0.000, E1   +48.934, E3 +309774.059}
SPL {X  -156.496, Y  +335.563, Z    +0.000, E1   +48.599, E3 +309783.636}
SPL {X  -154.894, Y  +330.318, Z    +0.000, E1   +48.380, E3 +309794.179}
SPL {X  -153.352, Y  +325.786, Z    +0.000, E1   +48.028, E3 +309803.935}
SPL {X  -151.316, Y  +320.384, Z    +0.000, E1   +47.734, E3 +309815.151}
SPL {X  -145.123, Y  +306.679, Z    +0.000, E1   +50.518, E3 +309823.966}
SPL {X  -135.207, Y  +289.783, Z    +0.000, E1   +44.101, E3 +309917.480}
ENDSPLINE

SPLINE
SPL {X  -154.528, Y  +329.203, Z    +0.000, E1   +28.834, E3 +309987.841}
SPL {X  -160.380, Y  +352.419, Z    +0.000, E1   +18.163, E3 +309992.202}
SPL {X  -162.408, Y  +368.921, Z    +0.000, E1    +9.337, E3 +309990.952}
SPL {X  -162.817, Y  +379.558, Z    +0.000, E1    +2.744, E3 +309991.342}
SPL {X  -162.820, Y  +384.383, Z    +0.000, E1    -0.869, E3 +309991.312}
SPL {X  -162.820, Y  +388.871, Z    +0.000, E1    -5.151, E3 +309991.017}
SPL {X  -162.820, Y  +395.861, Z    +0.000, E1   -13.028, E3 +309991.129}
SPL {X  -162.820, Y  +409.049, Z    +0.000, E1   -29.128, E3 +309989.971}
SPL {X  -162.820, Y  +444.592, Z    +0.000, E1   -49.032, E3 +310008.981}
SPL {X  -162.820, Y  +458.217, Z    +0.000, E1   -51.268, E3 +310020.926}
SPL {X  -162.820, Y  +501.848, Z    +0.000, E1   -54.235, E3 +310067.294}
ENDSPLINE

SPLINE
SPL {X  -162.820, Y  +498.156, Z    +0.000, E1   -50.986, E3 +310080.843}
ENDSPLINE

SPLINE
SPL {X  -162.820, Y  +499.429, Z    +0.000, E1   -49.453, E3 +310092.202}
SPL {X  -162.820, Y  +505.173, Z    +0.000, E1   -49.386, E3 +310102.857}
SPL {X  -162.820, Y  +510.642, Z    +0.000, E1   -49.447, E3 +310112.207}
SPL {X  -162.820, Y  +516.435, Z    +0.000, E1   -49.526, E3 +310122.085}
SPL {X  -162.820, Y  +523.383, Z    +0.000, E1   -49.407, E3 +310135.272}
SPL {X  -162.820, Y  +532.283, Z    +0.000, E1   -49.462, E3 +310150.875}
SPL {X  -162.820, Y  +541.471, Z    +0.000, E1   -49.456, E3 +310167.253}
SPL {X  -162.820, Y  +548.933, Z    +0.000, E1   -49.456, E3 +310180.441}
SPL {X  -162.820, Y  +553.997, Z    +0.000, E1   -49.325, E3 +310190.245}
SPL {X  -162.820, Y  +562.346, Z    +0.000, E1   -49.498, E3 +310204.307}
SPL {X  -162.820, Y  +570.444, Z    +0.000, E1   -49.421, E3 +310219.054}
SPL {X  -162.820, Y  +577.429, Z    +0.000, E1   -49.474, E3 +310231.168}
SPL {X  -162.820, Y  +585.965, Z    +0.000, E1   -49.447, E3 +310246.742}
SPL {X  -162.820, Y  +594.192, Z    +0.000, E1   -49.325, E3 +310261.985}
SPL {X  -162.820, Y  +600.267, Z    +0.000, E1   -49.443, E3 +310272.074}
SPL {X  -162.820, Y  +606.218, Z    +0.000, E1   -49.464, E3 +310282.621}
SPL {X  -162.820, Y  +612.538, Z    +0.000, E1   -49.488, E3 +310293.672}
SPL {X  -162.820, Y  +617.738, Z    +0.000, E1   -49.301, E3 +310304.108}
SPL {X  -162.820, Y  +624.265, Z    +0.000, E1   -49.443, E3 +310314.903}
SPL {X  -162.820, Y  +632.551, Z    +0.000, E1   -49.478, E3 +310329.672}
SPL {X  -162.820, Y  +641.207, Z    +0.000, E1   -49.420, E3 +310345.315}
SPL {X  -162.820, Y  +648.011, Z    +0.000, E1   -49.484, E3 +310356.992}
SPL {X  -162.820, Y  +655.976, Z    +0.000, E1   -49.445, E3 +310371.621}
SPL {X  -162.820, Y  +663.916, Z    +0.000, E1   -49.371, E3 +310386.050}
SPL {X  -162.820, Y  +669.755, Z    +0.000, E1   -49.387, E3 +310396.375}
SPL {X  -162.807, Y  +675.597, Z    +0.000, E1   -49.472, E3 +310406.277}
SPL {X  -162.632, Y  +681.322, Z    +0.000, E1   -49.345, E3 +310417.289}
SPL {X  -162.228, Y  +687.372, Z    +0.000, E1   -49.294, E3 +310428.375}
SPL {X  -161.723, Y  +692.372, Z    +0.000, E1   -49.172, E3 +310438.006}
SPL {X  -161.009, Y  +697.714, Z    +0.000, E1   -49.214, E3 +310447.290}
SPL {X  -160.313, Y  +701.965, Z    +0.000, E1   -48.932, E3 +310456.502}
SPL {X  -158.980, Y  +708.651, Z    +0.000, E1   -48.774, E3 +310469.542}
SPL {X  -157.477, Y  +714.869, Z    +0.000, E1   -48.424, E3 +310482.417}
SPL {X  -156.071, Y  +719.891, Z    +0.000, E1   -48.264, E3 +310492.294}
SPL {X  -154.661, Y  +724.395, Z    +0.000, E1   -47.951, E3 +310501.975}
SPL {X  -153.094, Y  +728.931, Z    +0.000, E1   -47.705, E3 +310511.412}
SPL {X  -151.300, Y  +733.655, Z    +0.000, E1   -47.339, E3 +310521.720}
SPL {X  -145.669, Y  +746.239, Z    +0.000, E1   -50.198, E3 +310528.497}
SPL {X  -135.084, Y  +764.399, Z    +0.000, E1   -44.787, E3 +310611.400}
ENDSPLINE

SPLINE
SPL {X  -153.038, Y  +729.086, Z    +0.000, E1   -30.522, E3 +310682.107}
SPL {X  -160.383, Y  +701.564, Z    +0.000, E1   -18.145, E3 +310692.143}
SPL {X  -162.078, Y  +689.023, Z    +0.000, E1   -11.510, E3 +310691.681}
SPL {X  -162.685, Y  +680.136, Z    +0.000, E1    -6.379, E3 +310691.970}
SPL {X  -162.820, Y  +672.919, Z    +0.000, E1    -1.752, E3 +310692.009}
SPL {X  -162.820, Y  +667.861, Z    +0.000, E1    +2.254, E3 +310691.810}
SPL {X  -162.820, Y  +662.755, Z    +0.000, E1    +7.521, E3 +310691.851}
SPL {X  -162.820, Y  +657.537, Z    +0.000, E1   +13.540, E3 +310691.520}
SPL {X  -162.820, Y  +650.460, Z    +0.000, E1   +22.200, E3 +310690.951}
SPL {X  -162.820, Y  +637.843, Z    +0.000, E1   +35.051, E3 +310693.028}
SPL {X  -162.820, Y  +595.072, Z    +0.000, E1   +53.652, E3 +310713.748}
SPL {X  -162.820, Y  +560.706, Z    +0.000, E1   +50.482, E3 +310774.657}
ENDSPLINE

SPLINE
SPL {X  -162.820, Y  +560.978, Z    +0.000, E1   +48.448, E3 +310786.743}
ENDSPLINE

SPLINE
SPL {X  -162.820, Y  +552.125, Z    +0.000, E1   +48.477, E3 +310802.848}
SPL {X  -162.820, Y  +545.800, Z    +0.000, E1   +48.334, E3 +310815.289}
SPL {X  -162.820, Y  +540.645, Z    +0.000, E1   +48.364, E3 +310824.640}
SPL {X  -162.820, Y  +534.689, Z    +0.000, E1   +48.295, E3 +310836.189}
SPL {X  -162.820, Y  +526.053, Z    +0.000, E1   +48.382, E3 +310851.764}
SPL {X  -162.820, Y  +519.666, Z    +0.000, E1   +48.261, E3 +310864.133}
SPL {X  -162.820, Y  +513.750, Z    +0.000, E1   +48.520, E3 +310873.575}
SPL {X  -162.820, Y  +508.282, Z    +0.000, E1   +48.307, E3 +310884.977}
SPL {X  -162.820, Y  +502.890, Z    +0.000, E1   +48.309, E3 +310894.904}
ENDSPLINE

SPLINE
SPL {X  -162.820, Y  +520.386, Z    +0.000, E1   +40.911, E3 +310901.634}
ENDSPLINE

SPLINE
SPL {X  -162.820, Y  +515.876, Z    +0.000, E1   +41.348, E3 +310909.832}
SPL {X  -162.820, Y  +507.007, Z    +0.000, E1   +42.470, E3 +310923.846}
SPL {X  -162.820, Y  +496.780, Z    +0.000, E1   +43.573, E3 +310940.101}
SPL {X  -162.820, Y  +488.962, Z    +0.000, E1   +44.342, E3 +310952.369}
SPL {X  -162.820, Y  +481.373, Z    +0.000, E1   +45.107, E3 +310963.853}
SPL {X  -162.820, Y  +473.909, Z    +0.000, E1   +45.743, E3 +310975.366}
SPL {X  -162.820, Y  +465.836, Z    +0.000, E1   +46.727, E3 +310985.657}
SPL {X  -162.820, Y  +457.217, Z    +0.000, E1   +47.671, E3 +310996.695}
SPL {X  -162.820, Y  +449.104, Z    +0.000, E1   +48.459, E3 +311007.163}
SPL {X  -162.820, Y  +440.303, Z    +0.000, E1   +49.204, E3 +311018.800}
SPL {X  -162.820, Y  +430.072, Z    +0.000, E1   +49.865, E3 +311033.102}
SPL {X  -162.820, Y  +423.062, Z    +0.000, E1   +49.728, E3 +311046.096}
SPL {X  -162.820, Y  +416.560, Z    +0.000, E1   +49.816, E3 +311057.077}
SPL {X  -162.820, Y  +410.559, Z    +0.000, E1   +49.727, E3 +311068.132}
SPL {X  -162.820, Y  +405.170, Z    +0.000, E1   +49.772, E3 +311077.334}
SPL {X  -162.820, Y  +398.766, Z    +0.000, E1   +49.793, E3 +311088.621}
SPL {X  -162.820, Y  +391.831, Z    +0.000, E1   +49.801, E3 +311100.667}
SPL {X  -162.820, Y  +386.334, Z    +0.000, E1   +49.739, E3 +311110.756}
SPL {X  -162.820, Y  +381.297, Z    +0.000, E1   +49.665, E3 +311120.027}
SPL {X  -162.709, Y  +374.487, Z    +0.000, E1   +49.773, E3 +311131.552}
SPL {X  -162.299, Y  +367.483, Z    +0.000, E1   +49.784, E3 +311143.694}
SPL {X  -161.760, Y  +361.947, Z    +0.000, E1   +49.515, E3 +311155.102}
SPL {X  -160.828, Y  +355.106, Z    +0.000, E1   +49.536, E3 +311167.019}
SPL {X  -159.832, Y  +349.452, Z    +0.000, E1   +49.188, E3 +311178.990}
SPL {X  -158.863, Y  +344.823, Z    +0.000, E1   +49.020, E3 +311188.039}
SPL {X  -157.695, Y  +339.971, Z    +0.000, E1   +48.934, E3 +311197.135}
SPL {X  -156.136, Y  +334.326, Z    +0.000, E1   +48.578, E3 +311209.102}
SPL {X  -154.561, Y  +329.302, Z    +0.000, E1   +48.290, E3 +311219.432}
SPL {X  -152.787, Y  +324.229, Z    +0.000, E1   +47.981, E3 +311230.123}
SPL {X  -150.789, Y  +319.074, Z    +0.000, E1   +47.585, E3 +311241.145}
SPL {X  -146.468, Y  +309.385, Z    +0.000, E1   +50.134, E3 +311244.691}
SPL {X  -143.047, Y  +302.732, Z    +0.000, E1   +51.043, E3 +311250.550}
SPL {X  -135.207, Y  +289.783, Z    +0.000, E1   +44.101, E3 +311340.557}
ENDSPLINE

SPLINE
SPL {X  -154.528, Y  +329.203, Z    +0.000, E1   +28.834, E3 +311410.918}
SPL {X  -160.380, Y  +352.419, Z    +0.000, E1   +18.163, E3 +311415.278}
SPL {X  -162.149, Y  +365.734, Z    +0.000, E1   +11.090, E3 +311413.887}
SPL {X  -162.754, Y  +375.862, Z    +0.000, E1    +5.134, E3 +311414.724}
SPL {X  -162.820, Y  +382.085, Z    +0.000, E1    +0.928, E3 +311414.413}
SPL {X  -162.820, Y  +386.028, Z    +0.000, E1    -2.328, E3 +311414.137}
SPL {X  -162.820, Y  +389.792, Z    +0.000, E1    -6.211, E3 +311414.069}
SPL {X  -162.820, Y  +395.861, Z    +0.000, E1   -13.028, E3 +311414.205}
SPL {X  -162.820, Y  +409.049, Z    +0.000, E1   -29.128, E3 +311413.048}
SPL {X  -162.820, Y  +444.592, Z    +0.000, E1   -49.032, E3 +311432.058}
SPL {X  -162.820, Y  +458.217, Z    +0.000, E1   -51.268, E3 +311444.003}
SPL {X  -162.820, Y  +501.848, Z    +0.000, E1   -54.235, E3 +311490.371}
ENDSPLINE

SPLINE
SPL {X  -162.820, Y  +498.156, Z    +0.000, E1   -50.986, E3 +311503.920}
ENDSPLINE

SPLINE
SPL {X  -162.820, Y  +499.429, Z    +0.000, E1   -49.453, E3 +311515.279}
SPL {X  -162.820, Y  +505.173, Z    +0.000, E1   -49.386, E3 +311525.934}
SPL {X  -162.820, Y  +510.642, Z    +0.000, E1   -49.447, E3 +311535.284}
SPL {X  -162.820, Y  +516.435, Z    +0.000, E1   -49.526, E3 +311545.162}
SPL {X  -162.820, Y  +522.095, Z    +0.000, E1   -49.420, E3 +311555.859}
SPL {X  -162.820, Y  +529.397, Z    +0.000, E1   -49.440, E3 +311568.868}
SPL {X  -162.820, Y  +536.932, Z    +0.000, E1   -49.395, E3 +311582.508}
SPL {X  -162.820, Y  +543.021, Z    +0.000, E1   -49.432, E3 +311593.114}
SPL {X  -162.820, Y  +548.933, Z    +0.000, E1   -49.456, E3 +311603.518}
SPL {X  -162.820, Y  +553.997, Z    +0.000, E1   -49.325, E3 +311613.322}
SPL {X  -162.820, Y  +560.268, Z    +0.000, E1   -49.531, E3 +311623.280}
SPL {X  -162.820, Y  +564.590, Z    +0.000, E1   -49.361, E3 +311631.980}
SPL {X  -162.820, Y  +570.444, Z    +0.000, E1   -49.421, E3 +311642.131}
SPL {X  -162.820, Y  +577.429, Z    +0.000, E1   -49.474, E3 +311654.245}
SPL {X  -162.820, Y  +582.387, Z    +0.000, E1   -49.269, E3 +311664.267}
SPL {X  -162.820, Y  +588.456, Z    +0.000, E1   -49.496, E3 +311673.781}
SPL {X  -162.820, Y  +594.192, Z    +0.000, E1   -49.325, E3 +311685.062}
SPL {X  -162.820, Y  +600.267, Z    +0.000, E1   -49.443, E3 +311695.151}
SPL {X  -162.820, Y  +606.218, Z    +0.000, E1   -49.464, E3 +311705.698}
SPL {X  -162.820, Y  +612.538, Z    +0.000, E1   -49.488, E3 +311716.749}
SPL {X  -162.820, Y  +617.738, Z    +0.000, E1   -49.301, E3 +311727.185}
SPL {X  -162.820, Y  +624.265, Z    +0.000, E1   -49.443, E3 +311737.980}
SPL {X  -162.820, Y  +630.226, Z    +0.000, E1   -49.472, E3 +311748.429}
SPL {X  -162.820, Y  +635.239, Z    +0.000, E1   -49.373, E3 +311757.924}
SPL {X  -162.820, Y  +641.207, Z    +0.000, E1   -49.420, E3 +311768.392}
SPL {X  -162.820, Y  +649.864, Z    +0.000, E1   -49.433, E3 +311783.871}
SPL {X  -162.820, Y  +658.147, Z    +0.000, E1   -49.491, E3 +311798.137}
SPL {X  -162.820, Y  +663.916, Z    +0.000, E1   -49.371, E3 +311809.127}
SPL {X  -162.820, Y  +669.755, Z    +0.000, E1   -49.387, E3 +311819.452}
SPL {X  -162.807, Y  +675.597, Z    +0.000, E1   -49.472, E3 +311829.354}
SPL {X  -162.632, Y  +681.322, Z    +0.000, E1   -49.345, E3 +311840.366}
SPL {X  -162.228, Y  +687.372, Z    +0.000, E1   -49.294, E3 +311851.452}
SPL {X  -161.723, Y  +692.372, Z    +0.000, E1   -49.172, E3 +311861.083}
SPL {X  -161.009, Y  +697.714, Z    +0.000, E1   -49.214, E3 +311870.367}
SPL {X  -160.313, Y  +701.965, Z    +0.000, E1   -48.932, E3 +311879.579}
SPL {X  -159.435, Y  +706.528, Z    +0.000, E1   -48.764, E3 +311888.706}
SPL {X  -157.894, Y  +713.249, Z    +0.000, E1   -48.586, E3 +311901.900}
SPL {X  -156.071, Y  +719.891, Z    +0.000, E1   -48.264, E3 +311915.371}
SPL {X  -154.661, Y  +724.395, Z    +0.000, E1   -47.951, E3 +311925.052}
SPL {X  -153.094, Y  +728.931, Z    +0.000, E1   -47.705, E3 +311934.489}
SPL {X  -151.300, Y  +733.655, Z    +0.000, E1   -47.339, E3 +311944.797}
SPL {X  -145.669, Y  +746.239, Z    +0.000, E1   -50.198, E3 +311951.573}
SPL {X  -135.084, Y  +764.399, Z    +0.000, E1   -44.787, E3 +312034.477}
ENDSPLINE

SPLINE
SPL {X  -153.038, Y  +729.086, Z    +0.000, E1   -30.522, E3 +312105.184}
SPL {X  -160.383, Y  +701.564, Z    +0.000, E1   -18.145, E3 +312115.220}
SPL {X  -162.078, Y  +689.023, Z    +0.000, E1   -11.510, E3 +312114.758}
SPL {X  -162.685, Y  +680.136, Z    +0.000, E1    -6.379, E3 +312115.047}
SPL {X  -162.820, Y  +672.919, Z    +0.000, E1    -1.752, E3 +312115.086}
SPL {X  -162.820, Y  +667.861, Z    +0.000, E1    +2.254, E3 +312114.887}
SPL {X  -162.820, Y  +662.755, Z    +0.000, E1    +7.521, E3 +312114.928}
SPL {X  -162.820, Y  +657.537, Z    +0.000, E1   +13.540, E3 +312114.597}
SPL {X  -162.820, Y  +650.460, Z    +0.000, E1   +22.200, E3 +312114.028}
SPL {X  -162.820, Y  +637.843, Z    +0.000, E1   +35.051, E3 +312116.105}
SPL {X  -162.820, Y  +595.072, Z    +0.000, E1   +53.652, E3 +312136.825}
SPL {X  -162.820, Y  +561.831, Z    +0.000, E1   +49.171, E3 +312204.048}
SPL {X  -162.820, Y  +555.289, Z    +0.000, E1   +48.406, E3 +312220.509}
SPL {X  -162.820, Y  +547.003, Z    +0.000, E1   +48.390, E3 +312235.921}
SPL {X  -162.820, Y  +540.645, Z    +0.000, E1   +48.364, E3 +312247.717}
SPL {X  -162.820, Y  +534.689, Z    +0.000, E1   +48.295, E3 +312259.266}
SPL {X  -162.820, Y  +528.564, Z    +0.000, E1   +48.407, E3 +312269.839}
SPL {X  -162.820, Y  +522.157, Z    +0.000, E1   +48.326, E3 +312282.420}
SPL {X  -162.820, Y  +513.750, Z    +0.000, E1   +48.520, E3 +312296.652}
SPL {X  -162.820, Y  +508.282, Z    +0.000, E1   +48.307, E3 +312308.054}
SPL {X  -162.820, Y  +502.890, Z    +0.000, E1   +48.309, E3 +312317.981}
ENDSPLINE

SPLINE
SPL {X  -162.820, Y  +517.326, Z    +0.000, E1   +41.232, E3 +312330.245}
ENDSPLINE

SPLINE
SPL {X  -162.820, Y  +507.007, Z    +0.000, E1   +42.470, E3 +312346.923}
SPL {X  -162.820, Y  +496.780, Z    +0.000, E1   +43.573, E3 +312363.178}
SPL {X  -162.820, Y  +488.962, Z    +0.000, E1   +44.342, E3 +312375.446}
SPL {X  -162.820, Y  +481.373, Z    +0.000, E1   +45.107, E3 +312386.930}
SPL {X  -162.820, Y  +473.909, Z    +0.000, E1   +45.743, E3 +312398.443}
SPL {X  -162.820, Y  +463.464, Z    +0.000, E1   +47.025, E3 +312411.660}
SPL {X  -162.820, Y  +451.336, Z    +0.000, E1   +48.248, E3 +312427.430}
SPL {X  -162.820, Y  +440.303, Z    +0.000, E1   +49.204, E3 +312441.877}
SPL {X  -162.820, Y  +430.072, Z    +0.000, E1   +49.865, E3 +312456.179}
SPL {X  -162.820, Y  +420.882, Z    +0.000, E1   +49.790, E3 +312472.790}
SPL {X  -162.820, Y  +411.982, Z    +0.000, E1   +49.786, E3 +312488.472}
SPL {X  -162.820, Y  +405.170, Z    +0.000, E1   +49.772, E3 +312500.411}
SPL {X  -162.820, Y  +398.766, Z    +0.000, E1   +49.793, E3 +312511.698}
SPL {X  -162.820, Y  +391.831, Z    +0.000, E1   +49.801, E3 +312523.744}
SPL {X  -162.820, Y  +384.205, Z    +0.000, E1   +49.756, E3 +312537.676}
SPL {X  -162.709, Y  +374.487, Z    +0.000, E1   +49.773, E3 +312554.628}
SPL {X  -162.197, Y  +366.269, Z    +0.000, E1   +49.717, E3 +312569.427}
SPL {X  -161.614, Y  +360.718, Z    +0.000, E1   +49.491, E3 +312580.412}
SPL {X  -160.828, Y  +355.106, Z    +0.000, E1   +49.536, E3 +312590.096}
SPL {X  -159.832, Y  +349.452, Z    +0.000, E1   +49.188, E3 +312602.067}
SPL {X  -158.863, Y  +344.823, Z    +0.000, E1   +49.020, E3 +312611.116}
SPL {X  -157.695, Y  +339.971, Z    +0.000, E1   +48.934, E3 +312620.212}
SPL {X  -156.136, Y  +334.326, Z    +0.000, E1   +48.578, E3 +312632.179}
SPL {X  -154.561, Y  +329.302, Z    +0.000, E1   +48.290, E3 +312642.509}
SPL {X  -153.352, Y  +325.786, Z    +0.000, E1   +48.028, E3 +312650.089}
SPL {X  -151.655, Y  +321.245, Z    +0.000, E1   +47.770, E3 +312659.510}
SPL {X  -150.383, Y  +318.088, Z    +0.000, E1   +47.517, E3 +312666.249}
SPL {X  -145.123, Y  +306.679, Z    +0.000, E1   +50.518, E3 +312670.119}
SPL {X  -135.207, Y  +289.783, Z    +0.000, E1   +44.101, E3 +312763.634}
ENDSPLINE

SPLINE
SPL {X  -154.528, Y  +329.203, Z    +0.000, E1   +28.834, E3 +312833.995}
SPL {X  -160.380, Y  +352.419, Z    +0.000, E1   +18.163, E3 +312838.355}
SPL {X  -162.408, Y  +368.921, Z    +0.000, E1    +9.337, E3 +312837.105}
SPL {X  -162.817, Y  +379.558, Z    +0.000, E1    +2.744, E3 +312837.495}
SPL {X  -162.820, Y  +384.383, Z    +0.000, E1    -0.869, E3 +312837.466}
SPL {X  -162.820, Y  +388.871, Z    +0.000, E1    -5.151, E3 +312837.171}
SPL {X  -162.820, Y  +395.861, Z    +0.000, E1   -13.028, E3 +312837.282}
SPL {X  -162.820, Y  +409.049, Z    +0.000, E1   -29.128, E3 +312836.125}
SPL {X  -162.820, Y  +446.299, Z    +0.000, E1   -49.360, E3 +312856.629}
SPL {X  -162.820, Y  +502.427, Z    +0.000, E1   -53.345, E3 +312919.614}
ENDSPLINE

SPLINE
SPL {X  -162.820, Y  +497.758, Z    +0.000, E1   -49.444, E3 +312935.553}
ENDSPLINE

